KUKA KRL program: MyProgram_028().src

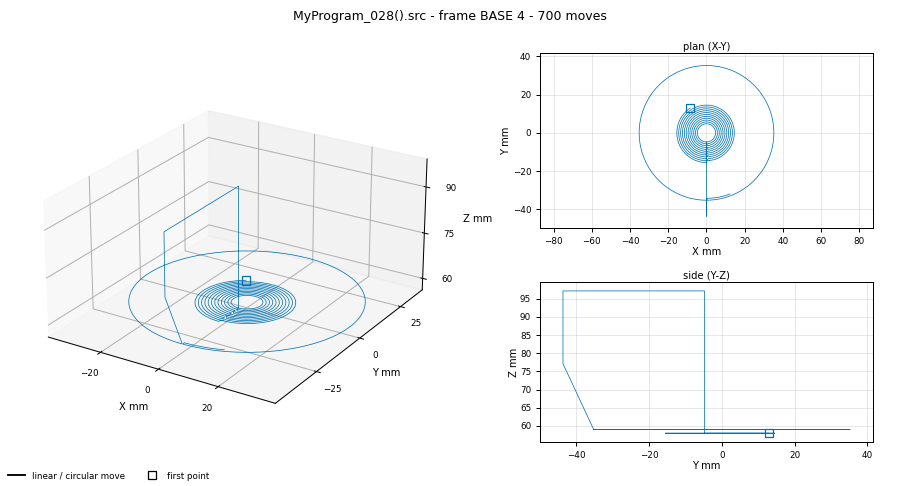
[picture p0: tool path of MyProgram_028().src in frame BASE 4, 700 of 700 moves have a stored position in this frame; points joined in program order, loops and branches not executed]
&ACCESS RVP
&REL 1
&PARAM TEMPLATE = C:\KRC\Roboter\Template\vorgabe
&PARAM EDITMASK = *
DEF MyProgram_028()
; ---- Setting reference (Base) ----
$BASE = BASE_DATA[4]

; --------------------------
; ---- Setting tool (TCP) ----
$TOOL = TOOL_DATA[3]
; --------------------------

$VEL.CP = VEL_APROX_PRINT
Startdeposition()
$VEL.CP = VEL_PRINT
LIN {X -8.4592,Y 13.0217,Z 58,A 116.025,B 24.784,C -3.3884,E1 24.9104,E2 -753.7985} C_DIS
LIN {X -9.3436,Y 12.4024,Z 58,A 119.821,B 24.785,C -3.3799,E1 24.9019,E2 -757.5875} C_DIS
LIN {X -10.555,Y 11.389,Z 58,A 127.1275,B 24.7861,C -3.3714,E1 24.8866,E2 -764.9027} C_DIS
LIN {X -12.1449,Y 9.676,Z 58,A 134.8717,B 24.7891,C -3.3477,E1 24.8724,E2 -772.6251} C_DIS
LIN {X -13.0597,Y 8.4004,Z 58,A 140.8782,B 24.791,C -3.3327,E1 24.863,E2 -778.6255} C_DIS
LIN {X -13.884,Y 6.9533,Z 58,A 146.3826,B 24.7934,C -3.3139,E1 24.8557,E2 -784.1139} C_DIS
LIN {X -14.682,Y 5.0559,Z 58,A 155.4146,B 24.7958,C -3.2945,E1 24.8466,E2 -793.15} C_DIS
LIN {X -15.1263,Y 3.5095,Z 58,A 161.5489,B 24.798,C -3.2767,E1 24.8426,E2 -799.2776} C_DIS
LIN {X -15.4979,Y 0.9698,Z 58,A 169.6776,B 24.802,C -3.2445,E1 24.8399,E2 -807.3778} C_DIS
LIN {X -15.5094,Y -0.7577,Z 58,A 177.1766,B 24.8041,C -3.2271,E1 24.8404,E2 -814.8801} C_DIS
LIN {X -15.3304,Y -2.4669,Z 58,A -177.0699,B 24.8066,C -3.2065,E1 24.8425,E2 -820.6186} C_DIS
LIN {X -14.8807,Y -4.4363,Z 58,A -169.0653,B 24.8091,C -3.1857,E1 24.8481,E2 -828.62} C_DIS
LIN {X -14.2177,Y -6.2434,Z 58,A -162.5125,B 24.8117,C -3.1645,E1 24.8549,E2 -835.1585} C_DIS
LIN {X -13.5937,Y -7.5059,Z 58,A -157.2385,B 24.8133,C -3.1509,E1 24.8617,E2 -840.428} C_DIS
LIN {X -13.0703,Y -8.3838,Z 58,A -153.3581,B 24.8144,C -3.1417,E1 24.8675,E2 -844.3061} C_DIS
LIN {X -12.191,Y -9.6177,Z 58,A -147.9234,B 24.816,C -3.1281,E1 24.8765,E2 -849.7344} C_DIS
LIN {X -11.3344,Y -10.6139,Z 58,A -142.9296,B 24.8172,C -3.1181,E1 24.8859,E2 -854.7263} C_DIS
LIN {X -10.3849,Y -11.5443,Z 58,A -138.2574,B 24.8184,C -3.1077,E1 24.8954,E2 -859.3928} C_DIS
LIN {X -9.5042,Y -12.2798,Z 58,A -134.1021,B 24.8193,C -3.0999,E1 24.9044,E2 -863.5451} C_DIS
LIN {X -8.6459,Y -12.8987,Z 58,A -129.7163,B 24.8199,C -3.0955,E1 24.9145,E2 -867.9351} C_DIS
LIN {X -7.2387,Y -13.7372,Z 58,A -123.8287,B 24.8209,C -3.0868,E1 24.9288,E2 -873.8193} C_DIS
LIN {X -5.9661,Y -14.3362,Z 58,A -119.1209,B 24.8217,C -3.0793,E1 24.9408,E2 -878.5205} C_DIS
LIN {X -4.8871,Y -14.7392,Z 58,A -114.3265,B 24.8219,C -3.0782,E1 24.9534,E2 -883.3216} C_DIS
LIN {X -3.7292,Y -15.0736,Z 58,A -110.1391,B 24.8223,C -3.0744,E1 24.9647,E2 -887.5063} C_DIS
LIN {X -2.6637,Y -15.298,Z 58,A -106.0151,B 24.8224,C -3.0735,E1 24.976,E2 -891.6326} C_DIS
LIN {X -1.431,Y -15.462,Z 58,A -101.5005,B 24.8225,C -3.0725,E1 24.9885,E2 -896.1478} C_DIS
LIN {X -0.1238,Y -15.5276,Z 58,A -96.4869,B 24.8223,C -3.0741,E1 25.0026,E2 -901.166} C_DIS
LIN {X -0.1238,Y -15.5276,Z 58,A -96.4869,B 24.8223,C -3.0741,E1 25.0026,E2 -901.166} C_DIS
Enddeposition()
LIN {X 0.0388,Y -14.5401,Z 58,A -3.2619,B 0,C 0,E1 0.1598,E2 -989.9292} C_DIS
Startdeposition()
$VEL.CP = VEL_PRINT
LIN {X -0.9942,Y -14.5149,Z 58,A -3.299,B 0,C 0,E1 0.1598,E2 -989.9288} C_DIS
LIN {X -2.6115,Y -14.3127,Z 58,A -3.3494,B 0,C 0,E1 0.1598,E2 -989.9289} C_DIS
LIN {X -4.0303,Y -13.9797,Z 58,A -3.3871,B 0,C 0,E1 0.1598,E2 -989.929} C_DIS
LIN {X -5.6828,Y -13.3931,Z 58,A -3.4223,B 0,C 0,E1 0.1598,E2 -989.9292} C_DIS
LIN {X -6.9637,Y -12.7741,Z 58,A -3.4428,B 0,C 0,E1 0.1598,E2 -989.9292} C_DIS
LIN {X -7.8731,Y -12.2346,Z 58,A -3.4532,B 0,C 0,E1 0.1598,E2 -989.9292} C_DIS
LIN {X -8.8006,Y -11.5856,Z 58,A -3.4594,B 0,C 0,E1 0.1598,E2 -989.9292} C_DIS
LIN {X -9.7294,Y -10.8172,Z 58,A -3.4607,B 0,C 0,E1 0.1598,E2 -989.9293} C_DIS
LIN {X -10.709,Y -9.8483,Z 58,A -3.4553,B 0,C 0,E1 0.1598,E2 -989.9295} C_DIS
LIN {X -11.4555,Y -8.9691,Z 58,A -3.4453,B 0,C 0,E1 0.1598,E2 -989.9295} C_DIS
LIN {X -12.3224,Y -7.735,Z 58,A -3.4244,B 0,C 0,E1 0.1598,E2 -989.9298} C_DIS
LIN {X -12.8548,Y -6.8137,Z 58,A -3.405,B 0,C 0,E1 0.1598,E2 -989.9296} C_DIS
LIN {X -13.4241,Y -5.6094,Z 58,A -3.3749,B 0,C 0,E1 0.1598,E2 -989.9296} C_DIS
LIN {X -13.7652,Y -4.7105,Z 58,A -3.3496,B 0,C 0,E1 0.1598,E2 -989.9293} C_DIS
LIN {X -14.1358,Y -3.4425,Z 58,A -3.3092,B 0,C 0,E1 0.1598,E2 -989.9297} C_DIS
LIN {X -14.3481,Y -2.4084,Z 58,A -3.2735,B 0,C 0,E1 0.1598,E2 -989.9294} C_DIS
LIN {X -14.5106,Y -1.0563,Z 58,A -3.222,B 0,C 0,E1 0.1598,E2 -989.9296} C_DIS
LIN {X -14.5449,Y 0.3484,Z 58,A -3.1636,B 0,C 0,E1 0.1598,E2 -989.9298} C_DIS
LIN {X -14.4218,Y 1.9199,Z 58,A -3.0926,B 0,C 0,E1 0.1598,E2 -989.9298} C_DIS
LIN {X -14.1478,Y 3.3932,Z 58,A -3.0205,B 0,C 0,E1 0.1598,E2 -989.9295} C_DIS
LIN {X -13.7525,Y 4.7484,Z 58,A -2.9488,B 0,C 0,E1 0.1598,E2 -989.9293} C_DIS
LIN {X -13.1379,Y 6.2501,Z 58,A -2.8624,B 0,C 0,E1 0.1598,E2 -989.9296} C_DIS
LIN {X -12.3406,Y 7.706,Z 58,A -2.7718,B 0,C 0,E1 0.1598,E2 -989.9291} C_DIS
LIN {X -11.6841,Y 8.6682,Z 58,A -2.7074,B 0,C 0,E1 0.1598,E2 -989.9285} C_DIS
LIN {X -10.8295,Y 9.7157,Z 58,A -2.6316,B 0,C 0,E1 0.1598,E2 -989.9285} C_DIS
LIN {X -10.0623,Y 10.5075,Z 58,A -2.57,B 0,C 0,E1 0.1598,E2 -989.9282} C_DIS
LIN {X -9.0076,Y 11.4252,Z 58,A -2.4922,B 0,C 0,E1 0.1598,E2 -989.9282} C_DIS
LIN {X -8.1523,Y 12.0501,Z 58,A -2.4343,B 0,C 0,E1 0.1598,E2 -989.9279} C_DIS
LIN {X -6.8933,Y 12.8124,Z 58,A -2.3555,B 0,C 0,E1 0.1598,E2 -989.9279} C_DIS
LIN {X -4.9769,Y 13.6712,Z 58,A -2.2483,B 0,C 0,E1 0.1598,E2 -989.9276} C_DIS
LIN {X -3.235,Y 14.1848,Z 58,A -2.1622,B 0,C 0,E1 0.1598,E2 -989.9274} C_DIS
LIN {X -1.6001,Y 14.4606,Z 58,A -2.09,B 0,C 0,E1 0.1598,E2 -989.9273} C_DIS
LIN {X 0.9482,Y 14.518,Z 58,A -1.9933,B 0,C 0,E1 0.1598,E2 -989.9271} C_DIS
LIN {X 1.9003,Y 14.4243,Z 58,A -1.962,B 0,C 0,E1 0.1598,E2 -989.9271} C_DIS
LIN {X 3.5313,Y 14.114,Z 58,A -1.9147,B 0,C 0,E1 0.1598,E2 -989.9271} C_DIS
LIN {X 4.9251,Y 13.6899,Z 58,A -1.8811,B 0,C 0,E1 0.1598,E2 -989.9271} C_DIS
LIN {X 6.3243,Y 13.1023,Z 58,A -1.8542,B 0,C 0,E1 0.1598,E2 -989.9272} C_DIS
LIN {X 7.3749,Y 12.5407,Z 58,A -1.8393,B 0,C 0,E1 0.1598,E2 -989.9272} C_DIS
LIN {X 8.2076,Y 12.0129,Z 58,A -1.8311,B 0,C 0,E1 0.1598,E2 -989.9271} C_DIS
LIN {X 9.0246,Y 11.4118,Z 58,A -1.8265,B 0,C 0,E1 0.1598,E2 -989.9271} C_DIS
LIN {X 10.1139,Y 10.4585,Z 58,A -1.8265,B 0,C 0,E1 0.1598,E2 -989.9275} C_DIS
LIN {X 11.0798,Y 9.4291,Z 58,A -1.8348,B 0,C 0,E1 0.1598,E2 -989.9276} C_DIS
LIN {X 11.7038,Y 8.6426,Z 58,A -1.8456,B 0,C 0,E1 0.1598,E2 -989.9273} C_DIS
LIN {X 12.3735,Y 7.6532,Z 58,A -1.8631,B 0,C 0,E1 0.1598,E2 -989.9275} C_DIS
LIN {X 13.2023,Y 6.1131,Z 58,A -1.8975,B 0,C 0,E1 0.1598,E2 -989.9285} C_DIS
LIN {X 13.7467,Y 4.7638,Z 58,A -1.9355,B 0,C 0,E1 0.1598,E2 -989.9283} C_DIS
LIN {X 14.1968,Y 3.1829,Z 58,A -1.9865,B 0,C 0,E1 0.1598,E2 -989.9286} C_DIS
LIN {X 14.3842,Y 2.1828,Z 58,A -2.0233,B 0,C 0,E1 0.1598,E2 -989.9278} C_DIS
LIN {X 14.5141,Y 1.0069,Z 58,A -2.0688,B 0,C 0,E1 0.1598,E2 -989.928} C_DIS
LIN {X 14.5491,Y -0.1159,Z 58,A -2.1158,B 0,C 0,E1 0.1598,E2 -989.928} C_DIS
LIN {X 14.4896,Y -1.3124,Z 58,A -2.1693,B 0,C 0,E1 0.1598,E2 -989.9281} C_DIS
LIN {X 14.3373,Y -2.4736,Z 58,A -2.2248,B 0,C 0,E1 0.1598,E2 -989.9281} C_DIS
LIN {X 14.0339,Y -3.8372,Z 58,A -2.2941,B 0,C 0,E1 0.1598,E2 -989.9287} C_DIS
LIN {X 13.6044,Y -5.1566,Z 58,A -2.3662,B 0,C 0,E1 0.1598,E2 -989.929} C_DIS
LIN {X 12.9068,Y -6.7148,Z 58,A -2.4589,B 0,C 0,E1 0.1598,E2 -989.929} C_DIS
LIN {X 12.2499,Y -7.8494,Z 58,A -2.5322,B 0,C 0,E1 0.1598,E2 -989.9286} C_DIS
LIN {X 11.5407,Y -8.8591,Z 58,A -2.6018,B 0,C 0,E1 0.1598,E2 -989.9284} C_DIS
LIN {X 10.8727,Y -9.6672,Z 58,A -2.6611,B 0,C 0,E1 0.1598,E2 -989.9284} C_DIS
LIN {X 9.8554,Y -10.7025,Z 58,A -2.7426,B 0,C 0,E1 0.1598,E2 -989.9286} C_DIS
LIN {X 8.7875,Y -11.5949,Z 58,A -2.8201,B 0,C 0,E1 0.1598,E2 -989.9286} C_DIS
LIN {X 7.8619,Y -12.2418,Z 58,A -2.8819,B 0,C 0,E1 0.1598,E2 -989.9285} C_DIS
LIN {X 6.6936,Y -12.918,Z 58,A -2.9536,B 0,C 0,E1 0.1598,E2 -989.9286} C_DIS
LIN {X 5.5443,Y -13.4512,Z 58,A -3.0186,B 0,C 0,E1 0.1598,E2 -989.9286} C_DIS
LIN {X 4.2078,Y -13.9272,Z 58,A -3.0879,B 0,C 0,E1 0.1598,E2 -989.9286} C_DIS
LIN {X 2.8277,Y -14.2717,Z 58,A -3.1531,B 0,C 0,E1 0.1598,E2 -989.9286} C_DIS
LIN {X 1.6425,Y -14.456,Z 58,A -3.2043,B 0,C 0,E1 0.1598,E2 -989.9287} C_DIS
LIN {X 0.0388,Y -14.5401,Z 58,A -3.2665,B 0,C 0,E1 0.1598,E2 -989.9287} C_DIS
Enddeposition()
LIN {X 0.0388,Y -14.5401,Z 58,A -3.2665,B 0,C 0,E1 0.1598,E2 -989.9287} C_DIS
Startdeposition()
$VEL.CP = VEL_PRINT
LIN {X 0.8886,Y -13.5406,Z 58,A -3.1918,B 0,C 0,E1 0.1598,E2 -989.9293} C_DIS
LIN {X 3.2193,Y -13.1824,Z 58,A -3.0918,B 0,C 0,E1 0.1598,E2 -989.9286} C_DIS
LIN {X 4.9417,Y -12.638,Z 58,A -3.0054,B 0,C 0,E1 0.1598,E2 -989.9286} C_DIS
LIN {X 6.7484,Y -11.7728,Z 58,A -2.902,B 0,C 0,E1 0.1598,E2 -989.9286} C_DIS
LIN {X 7.9074,Y -11.0278,Z 58,A -2.8277,B 0,C 0,E1 0.1598,E2 -989.9286} C_DIS
LIN {X 9.1575,Y -10.014,Z 58,A -2.7383,B 0,C 0,E1 0.1598,E2 -989.9286} C_DIS
LIN {X 10.2881,Y -8.8486,Z 58,A -2.6466,B 0,C 0,E1 0.1598,E2 -989.9287} C_DIS
LIN {X 11.189,Y -7.6776,Z 58,A -2.5634,B 0,C 0,E1 0.1598,E2 -989.9285} C_DIS
LIN {X 12.0375,Y -6.2635,Z 58,A -2.4712,B 0,C 0,E1 0.1598,E2 -989.9288} C_DIS
LIN {X 12.5414,Y -5.181,Z 58,A -2.4065,B 0,C 0,E1 0.1598,E2 -989.9284} C_DIS
LIN {X 13.1248,Y -3.4468,Z 58,A -2.3098,B 0,C 0,E1 0.1598,E2 -989.9292} C_DIS
LIN {X 13.4758,Y -1.5941,Z 58,A -2.2168,B 0,C 0,E1 0.1598,E2 -989.9296} C_DIS
LIN {X 13.4758,Y -1.5941,Z 58,A -2.2178,B 0,C 0,E1 0.1598,E2 -989.9285} C_DIS
LIN {X 13.57,Y 0.0222,Z 58,A -2.1447,B 0,C 0,E1 0.1598,E2 -989.9287} C_DIS
LIN {X 13.4778,Y 1.5775,Z 58,A -2.0812,B 0,C 0,E1 0.1598,E2 -989.9288} C_DIS
LIN {X 13.2328,Y 3.0058,Z 58,A -2.0294,B 0,C 0,E1 0.1598,E2 -989.9283} C_DIS
LIN {X 12.7101,Y 4.7521,Z 58,A -1.9731,B 0,C 0,E1 0.1598,E2 -989.9289} C_DIS
LIN {X 12.2201,Y 5.8998,Z 58,A -1.943,B 0,C 0,E1 0.1598,E2 -989.9279} C_DIS
LIN {X 11.7305,Y 6.822,Z 58,A -1.9218,B 0,C 0,E1 0.1598,E2 -989.9276} C_DIS
LIN {X 10.999,Y 7.9474,Z 58,A -1.9004,B 0,C 0,E1 0.1598,E2 -989.9278} C_DIS
LIN {X 10.0869,Y 9.0771,Z 58,A -1.8858,B 0,C 0,E1 0.1598,E2 -989.9278} C_DIS
LIN {X 9.1239,Y 10.0413,Z 58,A -1.8804,B 0,C 0,E1 0.1598,E2 -989.9276} C_DIS
LIN {X 8.0971,Y 10.8894,Z 58,A -1.8822,B 0,C 0,E1 0.1598,E2 -989.9274} C_DIS
LIN {X 7.1861,Y 11.5108,Z 58,A -1.8896,B 0,C 0,E1 0.1598,E2 -989.9272} C_DIS
LIN {X 6.149,Y 12.0958,Z 58,A -1.9031,B 0,C 0,E1 0.1598,E2 -989.9272} C_DIS
LIN {X 5.1555,Y 12.5523,Z 58,A -1.9204,B 0,C 0,E1 0.1598,E2 -989.9272} C_DIS
LIN {X 3.88,Y 13.0033,Z 58,A -1.9484,B 0,C 0,E1 0.1598,E2 -989.9272} C_DIS
LIN {X 2.4255,Y 13.3513,Z 58,A -1.9875,B 0,C 0,E1 0.1598,E2 -989.9272} C_DIS
LIN {X 1.2335,Y 13.5136,Z 58,A -2.0248,B 0,C 0,E1 0.1598,E2 -989.9272} C_DIS
LIN {X 0.0205,Y 13.5698,Z 58,A -2.0673,B 0,C 0,E1 0.1598,E2 -989.9272} C_DIS
LIN {X -1.423,Y 13.495,Z 58,A -2.1239,B 0,C 0,E1 0.1598,E2 -989.9272} C_DIS
LIN {X -2.9166,Y 13.2527,Z 58,A -2.1894,B 0,C 0,E1 0.1598,E2 -989.9274} C_DIS
LIN {X -4.4178,Y 12.8306,Z 58,A -2.2628,B 0,C 0,E1 0.1598,E2 -989.9275} C_DIS
LIN {X -5.6902,Y 12.3192,Z 58,A -2.3315,B 0,C 0,E1 0.1598,E2 -989.9277} C_DIS
LIN {X -7.1276,Y 11.5468,Z 58,A -2.4172,B 0,C 0,E1 0.1598,E2 -989.9279} C_DIS
LIN {X -8.359,Y 10.6897,Z 58,A -2.4988,B 0,C 0,E1 0.1598,E2 -989.9281} C_DIS
LIN {X -10.1247,Y 9.035,Z 58,A -2.6337,B 0,C 0,E1 0.1598,E2 -989.9286} C_DIS
LIN {X -11.3705,Y 7.4059,Z 58,A -2.7477,B 0,C 0,E1 0.1598,E2 -989.9295} C_DIS
LIN {X -11.9137,Y 6.4965,Z 58,A -2.807,B 0,C 0,E1 0.1598,E2 -989.9287} C_DIS
LIN {X -12.4568,Y 5.3822,Z 58,A -2.8739,B 0,C 0,E1 0.1598,E2 -989.929} C_DIS
LIN {X -12.8799,Y 4.271,Z 58,A -2.9366,B 0,C 0,E1 0.1598,E2 -989.929} C_DIS
LIN {X -13.4389,Y 1.8798,Z 58,A -3.0559,B 0,C 0,E1 0.1598,E2 -989.9313} C_DIS
LIN {X -13.4389,Y 1.8798,Z 58,A -3.0574,B 0,C 0,E1 0.1598,E2 -989.9299} C_DIS
LIN {X -13.5701,Y -0.0445,Z 58,A -3.1435,B 0,C 0,E1 0.1598,E2 -989.9299} C_DIS
LIN {X -13.3426,Y -2.4729,Z 58,A -3.2364,B 0,C 0,E1 0.1598,E2 -989.9314} C_DIS
LIN {X -13.3426,Y -2.4729,Z 58,A -3.2378,B 0,C 0,E1 0.1598,E2 -989.93} C_DIS
LIN {X -13.0748,Y -3.632,Z 58,A -3.2776,B 0,C 0,E1 0.1598,E2 -989.9295} C_DIS
LIN {X -12.4435,Y -5.4128,Z 58,A -3.3289,B 0,C 0,E1 0.1598,E2 -989.9305} C_DIS
LIN {X -11.9464,Y -6.436,Z 58,A -3.3549,B 0,C 0,E1 0.1598,E2 -989.9296} C_DIS
LIN {X -11.4777,Y -7.2392,Z 58,A -3.3721,B 0,C 0,E1 0.1598,E2 -989.9292} C_DIS
LIN {X -10.8186,Y -8.1914,Z 58,A -3.3882,B 0,C 0,E1 0.1598,E2 -989.9294} C_DIS
LIN {X -10.0004,Y -9.1723,Z 58,A -3.3998,B 0,C 0,E1 0.1598,E2 -989.9294} C_DIS
LIN {X -8.8658,Y -10.2733,Z 58,A -3.4052,B 0,C 0,E1 0.1598,E2 -989.9294} C_DIS
LIN {X -7.8194,Y -11.0904,Z 58,A -3.4016,B 0,C 0,E1 0.1598,E2 -989.9293} C_DIS
LIN {X -6.1046,Y -12.1193,Z 58,A -3.3824,B 0,C 0,E1 0.1598,E2 -989.9295} C_DIS
LIN {X -4.9242,Y -12.6447,Z 58,A -3.362,B 0,C 0,E1 0.1598,E2 -989.9291} C_DIS
LIN {X -3.8579,Y -13.0098,Z 58,A -3.3386,B 0,C 0,E1 0.1598,E2 -989.929} C_DIS
LIN {X -1.3592,Y -13.5016,Z 58,A -3.2683,B 0,C 0,E1 0.1598,E2 -989.9289} C_DIS
LIN {X -0.3554,Y -13.5648,Z 58,A -3.2344,B 0,C 0,E1 0.1598,E2 -989.9287} C_DIS
LIN {X -0.3554,Y -13.5648,Z 58,A -3.2344,B 0,C 0,E1 0.1598,E2 -989.9287} C_DIS
Enddeposition()
LIN {X 0.0583,Y -12.5898,Z 58,A -3.1759,B 0,C 0,E1 0.1598,E2 -989.93} C_DIS
Startdeposition()
$VEL.CP = VEL_PRINT
LIN {X -1.1152,Y -12.5412,Z 58,A -3.218,B 0,C 0,E1 0.1598,E2 -989.9288} C_DIS
LIN {X -2.5157,Y -12.3362,Z 58,A -3.2605,B 0,C 0,E1 0.1598,E2 -989.9288} C_DIS
LIN {X -3.6853,Y -12.0392,Z 58,A -3.2906,B 0,C 0,E1 0.1598,E2 -989.9288} C_DIS
LIN {X -4.9903,Y -11.5595,Z 58,A -3.3178,B 0,C 0,E1 0.1598,E2 -989.929} C_DIS
LIN {X -6.4135,Y -10.8344,Z 58,A -3.3389,B 0,C 0,E1 0.1598,E2 -989.9292} C_DIS
LIN {X -7.4925,Y -10.1188,Z 58,A -3.3479,B 0,C 0,E1 0.1598,E2 -989.9292} C_DIS
LIN {X -8.3401,Y -9.4323,Z 58,A -3.3498,B 0,C 0,E1 0.1598,E2 -989.9292} C_DIS
LIN {X -9.2947,Y -8.4931,Z 58,A -3.3447,B 0,C 0,E1 0.1598,E2 -989.9294} C_DIS
LIN {X -10.0403,Y -7.5973,Z 58,A -3.3341,B 0,C 0,E1 0.1598,E2 -989.9293} C_DIS
LIN {X -10.6375,Y -6.7357,Z 58,A -3.3194,B 0,C 0,E1 0.1598,E2 -989.9293} C_DIS
LIN {X -11.4083,Y -5.3268,Z 58,A -3.2871,B 0,C 0,E1 0.1598,E2 -989.93} C_DIS
LIN {X -11.9956,Y -3.8248,Z 58,A -3.2449,B 0,C 0,E1 0.1598,E2 -989.93} C_DIS
LIN {X -12.298,Y -2.6958,Z 58,A -3.2089,B 0,C 0,E1 0.1598,E2 -989.9294} C_DIS
LIN {X -12.4965,Y -1.5381,Z 58,A -3.167,B 0,C 0,E1 0.1598,E2 -989.9294} C_DIS
LIN {X -12.5734,Y -0.6576,Z 58,A -3.1331,B 0,C 0,E1 0.1598,E2 -989.929} C_DIS
LIN {X -12.5492,Y 1.0206,Z 58,A -3.0601,B 0,C 0,E1 0.1598,E2 -989.9299} C_DIS
LIN {X -12.3016,Y 2.682,Z 58,A -2.9801,B 0,C 0,E1 0.1598,E2 -989.9305} C_DIS
LIN {X -12.3016,Y 2.682,Z 58,A -2.9812,B 0,C 0,E1 0.1598,E2 -989.9294} C_DIS
LIN {X -11.7711,Y 4.4677,Z 58,A -2.8856,B 0,C 0,E1 0.1598,E2 -989.9298} C_DIS
LIN {X -10.8953,Y 6.3101,Z 58,A -2.7753,B 0,C 0,E1 0.1598,E2 -989.9298} C_DIS
LIN {X -9.9971,Y 7.6532,Z 58,A -2.686,B 0,C 0,E1 0.1598,E2 -989.929} C_DIS
LIN {X -9.045,Y 8.7585,Z 58,A -2.6046,B 0,C 0,E1 0.1598,E2 -989.9285} C_DIS
LIN {X -8.1234,Y 9.6193,Z 58,A -2.5343,B 0,C 0,E1 0.1598,E2 -989.9282} C_DIS
LIN {X -6.7121,Y 10.6518,Z 58,A -2.4386,B 0,C 0,E1 0.1598,E2 -989.928} C_DIS
LIN {X -5.3838,Y 11.3817,Z 58,A -2.3586,B 0,C 0,E1 0.1598,E2 -989.9279} C_DIS
LIN {X -2.878,Y 12.2573,Z 58,A -2.2289,B 0,C 0,E1 0.1598,E2 -989.9276} C_DIS
LIN {X -1.0584,Y 12.5461,Z 58,A -2.1495,B 0,C 0,E1 0.1598,E2 -989.9273} C_DIS
LIN {X 0.828,Y 12.5633,Z 58,A -2.079,B 0,C 0,E1 0.1598,E2 -989.9273} C_DIS
LIN {X 2.6155,Y 12.3161,Z 58,A -2.0234,B 0,C 0,E1 0.1598,E2 -989.9272} C_DIS
LIN {X 4.8078,Y 11.6367,Z 58,A -1.9711,B 0,C 0,E1 0.1598,E2 -989.9272} C_DIS
LIN {X 6.468,Y 10.8023,Z 58,A -1.945,B 0,C 0,E1 0.1598,E2 -989.9275} C_DIS
LIN {X 7.714,Y 9.9507,Z 58,A -1.9352,B 0,C 0,E1 0.1598,E2 -989.9275} C_DIS
LIN {X 8.7384,Y 9.0644,Z 58,A -1.9352,B 0,C 0,E1 0.1598,E2 -989.9275} C_DIS
LIN {X 9.5305,Y 8.2277,Z 58,A -1.9418,B 0,C 0,E1 0.1598,E2 -989.9275} C_DIS
LIN {X 10.3825,Y 7.1226,Z 58,A -1.9571,B 0,C 0,E1 0.1598,E2 -989.9279} C_DIS
LIN {X 11.1706,Y 5.8084,Z 58,A -1.984,B 0,C 0,E1 0.1598,E2 -989.9283} C_DIS
LIN {X 11.7313,Y 4.5716,Z 58,A -2.0165,B 0,C 0,E1 0.1598,E2 -989.928} C_DIS
LIN {X 12.1241,Y 3.3953,Z 58,A -2.0524,B 0,C 0,E1 0.1598,E2 -989.928} C_DIS
LIN {X 12.4715,Y 1.7265,Z 58,A -2.1099,B 0,C 0,E1 0.1598,E2 -989.9294} C_DIS
LIN {X 12.4715,Y 1.7265,Z 58,A -2.1109,B 0,C 0,E1 0.1598,E2 -989.9283} C_DIS
LIN {X 12.588,Y -0.2518,Z 58,A -2.1904,B 0,C 0,E1 0.1598,E2 -989.9294} C_DIS
LIN {X 12.588,Y -0.2518,Z 58,A -2.1915,B 0,C 0,E1 0.1598,E2 -989.9284} C_DIS
LIN {X 12.2824,Y -2.7694,Z 58,A -2.3081,B 0,C 0,E1 0.1598,E2 -989.9312} C_DIS
LIN {X 12.2824,Y -2.7694,Z 58,A -2.3099,B 0,C 0,E1 0.1598,E2 -989.9294} C_DIS
LIN {X 11.4381,Y -5.2626,Z 58,A -2.4463,B 0,C 0,E1 0.1598,E2 -989.9311} C_DIS
LIN {X 11.4381,Y -5.2626,Z 58,A -2.448,B 0,C 0,E1 0.1598,E2 -989.9294} C_DIS
LIN {X 10.6512,Y -6.714,Z 58,A -2.5394,B 0,C 0,E1 0.1598,E2 -989.9292} C_DIS
LIN {X 9.8702,Y -7.8162,Z 58,A -2.616,B 0,C 0,E1 0.1598,E2 -989.9285} C_DIS
LIN {X 8.4163,Y -9.3643,Z 58,A -2.7357,B 0,C 0,E1 0.1598,E2 -989.9287} C_DIS
LIN {X 7.6804,Y -9.9766,Z 58,A -2.7893,B 0,C 0,E1 0.1598,E2 -989.9283} C_DIS
LIN {X 6.4247,Y -10.8281,Z 58,A -2.8716,B 0,C 0,E1 0.1598,E2 -989.9286} C_DIS
LIN {X 5.0678,Y -11.5254,Z 58,A -2.9512,B 0,C 0,E1 0.1598,E2 -989.9286} C_DIS
LIN {X 4.0136,Y -11.9336,Z 58,A -3.0074,B 0,C 0,E1 0.1598,E2 -989.9286} C_DIS
LIN {X 2.0202,Y -12.4275,Z 58,A -3.1014,B 0,C 0,E1 0.1598,E2 -989.9286} C_DIS
LIN {X 0.6281,Y -12.5751,Z 58,A -3.1587,B 0,C 0,E1 0.1598,E2 -989.9286} C_DIS
LIN {X 0.6281,Y -12.5751,Z 58,A -3.1587,B 0,C 0,E1 0.1598,E2 -989.9286} C_DIS
Enddeposition()
LIN {X 0.0659,Y -11.608,Z 58,A -3.1363,B 0,C 0,E1 0.1598,E2 -989.9299} C_DIS
Startdeposition()
$VEL.CP = VEL_PRINT
LIN {X 0.9358,Y -11.5737,Z 58,A -3.1043,B 0,C 0,E1 0.1598,E2 -989.9286} C_DIS
LIN {X 2.2027,Y -11.4005,Z 58,A -3.0506,B 0,C 0,E1 0.1598,E2 -989.9286} C_DIS
LIN {X 3.2368,Y -11.1509,Z 58,A -3.0021,B 0,C 0,E1 0.1598,E2 -989.9285} C_DIS
LIN {X 5.2781,Y -10.3423,Z 58,A -2.8926,B 0,C 0,E1 0.1598,E2 -989.9285} C_DIS
LIN {X 6.1433,Y -9.8531,Z 58,A -2.84,B 0,C 0,E1 0.1598,E2 -989.9283} C_DIS
LIN {X 7.1677,Y -9.1352,Z 58,A -2.7715,B 0,C 0,E1 0.1598,E2 -989.9285} C_DIS
LIN {X 8.2194,Y -8.2017,Z 58,A -2.6929,B 0,C 0,E1 0.1598,E2 -989.9285} C_DIS
LIN {X 9.05,Y -7.275,Z 58,A -2.6227,B 0,C 0,E1 0.1598,E2 -989.9284} C_DIS
LIN {X 9.8561,Y -6.1384,Z 58,A -2.5441,B 0,C 0,E1 0.1598,E2 -989.9286} C_DIS
LIN {X 10.3697,Y -5.2247,Z 58,A -2.4863,B 0,C 0,E1 0.1598,E2 -989.9282} C_DIS
LIN {X 10.9795,Y -3.7785,Z 58,A -2.4013,B 0,C 0,E1 0.1598,E2 -989.9288} C_DIS
LIN {X 11.3407,Y -2.492,Z 58,A -2.3331,B 0,C 0,E1 0.1598,E2 -989.9284} C_DIS
LIN {X 11.5401,Y -1.2855,Z 58,A -2.2741,B 0,C 0,E1 0.1598,E2 -989.9283} C_DIS
LIN {X 11.6111,Y -0.1232,Z 58,A -2.2217,B 0,C 0,E1 0.1598,E2 -989.9282} C_DIS
LIN {X 11.5726,Y 0.948,Z 58,A -2.1772,B 0,C 0,E1 0.1598,E2 -989.9282} C_DIS
LIN {X 11.4265,Y 2.0639,Z 58,A -2.1348,B 0,C 0,E1 0.1598,E2 -989.928} C_DIS
LIN {X 11.1563,Y 3.2192,Z 58,A -2.0952,B 0,C 0,E1 0.1598,E2 -989.928} C_DIS
LIN {X 10.5769,Y 4.7912,Z 58,A -2.0486,B 0,C 0,E1 0.1598,E2 -989.9286} C_DIS
LIN {X 9.8604,Y 6.1315,Z 58,A -2.0179,B 0,C 0,E1 0.1598,E2 -989.9283} C_DIS
LIN {X 8.9529,Y 7.394,Z 58,A -1.9975,B 0,C 0,E1 0.1598,E2 -989.9282} C_DIS
LIN {X 8.0596,Y 8.3584,Z 58,A -1.9898,B 0,C 0,E1 0.1598,E2 -989.9277} C_DIS
LIN {X 7.0675,Y 9.2128,Z 58,A -1.9901,B 0,C 0,E1 0.1598,E2 -989.9276} C_DIS
LIN {X 5.8926,Y 10.0051,Z 58,A -1.9997,B 0,C 0,E1 0.1598,E2 -989.9275} C_DIS
LIN {X 5.0221,Y 10.4692,Z 58,A -2.0124,B 0,C 0,E1 0.1598,E2 -989.9273} C_DIS
LIN {X 4.0673,Y 10.8757,Z 58,A -2.0304,B 0,C 0,E1 0.1598,E2 -989.9273} C_DIS
LIN {X 2.8081,Y 11.2667,Z 58,A -2.0603,B 0,C 0,E1 0.1598,E2 -989.9273} C_DIS
LIN {X 1.8789,Y 11.456,Z 58,A -2.0867,B 0,C 0,E1 0.1598,E2 -989.9273} C_DIS
LIN {X 1.1267,Y 11.5541,Z 58,A -2.1104,B 0,C 0,E1 0.1598,E2 -989.9273} C_DIS
LIN {X -0.1376,Y 11.6107,Z 58,A -2.1547,B 0,C 0,E1 0.1598,E2 -989.9273} C_DIS
LIN {X -2.0552,Y 11.4281,Z 58,A -2.2333,B 0,C 0,E1 0.1598,E2 -989.9274} C_DIS
LIN {X -3.6219,Y 11.0322,Z 58,A -2.308,B 0,C 0,E1 0.1598,E2 -989.9276} C_DIS
LIN {X -5.0899,Y 10.4365,Z 58,A -2.3874,B 0,C 0,E1 0.1598,E2 -989.9278} C_DIS
LIN {X -6.3171,Y 9.7423,Z 58,A -2.462,B 0,C 0,E1 0.1598,E2 -989.928} C_DIS
LIN {X -7.671,Y 8.7161,Z 58,A -2.5551,B 0,C 0,E1 0.1598,E2 -989.9284} C_DIS
LIN {X -8.9876,Y 7.3509,Z 58,A -2.6612,B 0,C 0,E1 0.1598,E2 -989.9288} C_DIS
LIN {X -10.1678,Y 5.6075,Z 58,A -2.7778,B 0,C 0,E1 0.1598,E2 -989.9297} C_DIS
LIN {X -10.6295,Y 4.6732,Z 58,A -2.8353,B 0,C 0,E1 0.1598,E2 -989.9287} C_DIS
LIN {X -10.9996,Y 3.7108,Z 58,A -2.8897,B 0,C 0,E1 0.1598,E2 -989.9287} C_DIS
LIN {X -11.367,Y 2.3701,Z 58,A -2.9594,B 0,C 0,E1 0.1598,E2 -989.9294} C_DIS
LIN {X -11.5634,Y 1.0517,Z 58,A -3.0225,B 0,C 0,E1 0.1598,E2 -989.9294} C_DIS
LIN {X -11.5968,Y -0.5835,Z 58,A -3.0924,B 0,C 0,E1 0.1598,E2 -989.9299} C_DIS
LIN {X -11.4579,Y -1.8811,Z 58,A -3.1426,B 0,C 0,E1 0.1598,E2 -989.9295} C_DIS
LIN {X -10.93,Y -3.9197,Z 58,A -3.2094,B 0,C 0,E1 0.1598,E2 -989.9297} C_DIS
LIN {X -10.1671,Y -5.6087,Z 58,A -3.2527,B 0,C 0,E1 0.1598,E2 -989.9301} C_DIS
LIN {X -9.4269,Y -6.7795,Z 58,A -3.2758,B 0,C 0,E1 0.1598,E2 -989.9295} C_DIS
LIN {X -8.6887,Y -7.7029,Z 58,A -3.2881,B 0,C 0,E1 0.1598,E2 -989.9295} C_DIS
LIN {X -7.6348,Y -8.7484,Z 58,A -3.2939,B 0,C 0,E1 0.1598,E2 -989.9294} C_DIS
LIN {X -6.6824,Y -9.4959,Z 58,A -3.2911,B 0,C 0,E1 0.1598,E2 -989.9291} C_DIS
LIN {X -5.4334,Y -10.2618,Z 58,A -3.2779,B 0,C 0,E1 0.1598,E2 -989.9291} C_DIS
LIN {X -4.3888,Y -10.7501,Z 58,A -3.2606,B 0,C 0,E1 0.1598,E2 -989.929} C_DIS
LIN {X -3.3702,Y -11.1117,Z 58,A -3.2388,B 0,C 0,E1 0.1598,E2 -989.9288} C_DIS
LIN {X -1.4769,Y -11.5171,Z 58,A -3.1868,B 0,C 0,E1 0.1598,E2 -989.9288} C_DIS
LIN {X -0.5139,Y -11.5974,Z 58,A -3.1551,B 0,C 0,E1 0.1598,E2 -989.9286} C_DIS
LIN {X -0.5139,Y -11.5974,Z 58,A -3.1551,B 0,C 0,E1 0.1598,E2 -989.9286} C_DIS
Enddeposition()
LIN {X 0.0689,Y -10.6297,Z 58,A -3.0908,B 0,C 0,E1 0.1598,E2 -989.9299} C_DIS
Startdeposition()
$VEL.CP = VEL_PRINT
LIN {X -1.1138,Y -10.5738,Z 58,A -3.133,B 0,C 0,E1 0.1598,E2 -989.9287} C_DIS
LIN {X -2.3366,Y -10.3695,Z 58,A -3.1691,B 0,C 0,E1 0.1598,E2 -989.9287} C_DIS
LIN {X -3.1763,Y -10.1468,Z 58,A -3.1903,B 0,C 0,E1 0.1598,E2 -989.9287} C_DIS
LIN {X -4.3953,Y -9.6813,Z 58,A -3.215,B 0,C 0,E1 0.1598,E2 -989.9288} C_DIS
LIN {X -5.5525,Y -9.0673,Z 58,A -3.2312,B 0,C 0,E1 0.1598,E2 -989.9289} C_DIS
LIN {X -6.4304,Y -8.4673,Z 58,A -3.2378,B 0,C 0,E1 0.1598,E2 -989.9289} C_DIS
LIN {X -7.3345,Y -7.6976,Z 58,A -3.2381,B 0,C 0,E1 0.1598,E2 -989.9291} C_DIS
LIN {X -8.4849,Y -6.4072,Z 58,A -3.2253,B 0,C 0,E1 0.1598,E2 -989.9292} C_DIS
LIN {X -9.0728,Y -5.5434,Z 58,A -3.21,B 0,C 0,E1 0.1598,E2 -989.9294} C_DIS
LIN {X -9.7569,Y -4.2247,Z 58,A -3.1789,B 0,C 0,E1 0.1598,E2 -989.9296} C_DIS
LIN {X -10.1537,Y -3.1538,Z 58,A -3.1484,B 0,C 0,E1 0.1598,E2 -989.9292} C_DIS
LIN {X -10.4297,Y -2.0648,Z 58,A -3.1124,B 0,C 0,E1 0.1598,E2 -989.9292} C_DIS
LIN {X -10.5922,Y -0.9234,Z 58,A -3.0698,B 0,C 0,E1 0.1598,E2 -989.9293} C_DIS
LIN {X -10.6324,Y 0.0112,Z 58,A -3.0321,B 0,C 0,E1 0.1598,E2 -989.9289} C_DIS
LIN {X -10.5469,Y 1.3416,Z 58,A -2.9721,B 0,C 0,E1 0.1598,E2 -989.9293} C_DIS
LIN {X -10.3722,Y 2.3358,Z 58,A -2.924,B 0,C 0,E1 0.1598,E2 -989.9289} C_DIS
LIN {X -10.0307,Y 3.5256,Z 58,A -2.8609,B 0,C 0,E1 0.1598,E2 -989.9289} C_DIS
LIN {X -9.4167,Y 4.9368,Z 58,A -2.7781,B 0,C 0,E1 0.1598,E2 -989.9293} C_DIS
LIN {X -8.0269,Y 6.9724,Z 58,A -2.6409,B 0,C 0,E1 0.1598,E2 -989.9289} C_DIS
LIN {X -6.7605,Y 8.2055,Z 58,A -2.5421,B 0,C 0,E1 0.1598,E2 -989.9286} C_DIS
LIN {X -6.013,Y 8.7688,Z 58,A -2.4912,B 0,C 0,E1 0.1598,E2 -989.928} C_DIS
LIN {X -5.2827,Y 9.227,Z 58,A -2.4449,B 0,C 0,E1 0.1598,E2 -989.9279} C_DIS
LIN {X -3.9678,Y 9.8643,Z 58,A -2.3693,B 0,C 0,E1 0.1598,E2 -989.9279} C_DIS
LIN {X -2.6913,Y 10.286,Z 58,A -2.3043,B 0,C 0,E1 0.1598,E2 -989.9276} C_DIS
LIN {X -1.198,Y 10.5646,Z 58,A -2.2374,B 0,C 0,E1 0.1598,E2 -989.9274} C_DIS
LIN {X 0.2712,Y 10.6289,Z 58,A -2.1804,B 0,C 0,E1 0.1598,E2 -989.9274} C_DIS
LIN {X 1.5071,Y 10.5226,Z 58,A -2.1392,B 0,C 0,E1 0.1598,E2 -989.9274} C_DIS
LIN {X 2.8024,Y 10.2563,Z 58,A -2.1026,B 0,C 0,E1 0.1598,E2 -989.9274} C_DIS
LIN {X 3.8876,Y 9.896,Z 58,A -2.0778,B 0,C 0,E1 0.1598,E2 -989.9274} C_DIS
LIN {X 4.702,Y 9.5359,Z 58,A -2.0631,B 0,C 0,E1 0.1598,E2 -989.9273} C_DIS
LIN {X 5.8089,Y 8.9053,Z 58,A -2.0489,B 0,C 0,E1 0.1598,E2 -989.9274} C_DIS
LIN {X 6.8841,Y 8.1028,Z 58,A -2.0433,B 0,C 0,E1 0.1598,E2 -989.9276} C_DIS
LIN {X 7.8782,Y 7.1403,Z 58,A -2.0475,B 0,C 0,E1 0.1598,E2 -989.9277} C_DIS
LIN {X 8.7786,Y 5.9985,Z 58,A -2.0628,B 0,C 0,E1 0.1598,E2 -989.928} C_DIS
LIN {X 9.3776,Y 5.0108,Z 58,A -2.0831,B 0,C 0,E1 0.1598,E2 -989.9279} C_DIS
LIN {X 9.74,Y 4.2636,Z 58,A -2.102,B 0,C 0,E1 0.1598,E2 -989.9276} C_DIS
LIN {X 10.3374,Y 2.4868,Z 58,A -2.1545,B 0,C 0,E1 0.1598,E2 -989.9292} C_DIS
LIN {X 10.6211,Y 0.4869,Z 58,A -2.2293,B 0,C 0,E1 0.1598,E2 -989.9297} C_DIS
LIN {X 10.6211,Y 0.4869,Z 58,A -2.2304,B 0,C 0,E1 0.1598,E2 -989.9285} C_DIS
LIN {X 10.5933,Y -0.9108,Z 58,A -2.2913,B 0,C 0,E1 0.1598,E2 -989.9286} C_DIS
LIN {X 10.4469,Y -1.9768,Z 58,A -2.3428,B 0,C 0,E1 0.1598,E2 -989.9282} C_DIS
LIN {X 10.1303,Y -3.2277,Z 58,A -2.4077,B 0,C 0,E1 0.1598,E2 -989.9287} C_DIS
LIN {X 9.6928,Y -4.3697,Z 58,A -2.473,B 0,C 0,E1 0.1598,E2 -989.9285} C_DIS
LIN {X 9.0572,Y -5.569,Z 58,A -2.5476,B 0,C 0,E1 0.1598,E2 -989.9287} C_DIS
LIN {X 8.5038,Y -6.3819,Z 58,A -2.6032,B 0,C 0,E1 0.1598,E2 -989.9282} C_DIS
LIN {X 7.0479,Y -7.9609,Z 58,A -2.7234,B 0,C 0,E1 0.1598,E2 -989.9292} C_DIS
LIN {X 5.4991,Y -9.0993,Z 58,A -2.8297,B 0,C 0,E1 0.1598,E2 -989.9285} C_DIS
LIN {X 3.9607,Y -9.867,Z 58,A -2.9191,B 0,C 0,E1 0.1598,E2 -989.9285} C_DIS
LIN {X 2.3268,Y -10.3747,Z 58,A -3.0006,B 0,C 0,E1 0.1598,E2 -989.9285} C_DIS
LIN {X 0.9025,Y -10.594,Z 58,A -3.0622,B 0,C 0,E1 0.1598,E2 -989.9285} C_DIS
LIN {X 0.0689,Y -10.6297,Z 58,A -3.0943,B 0,C 0,E1 0.1598,E2 -989.9285} C_DIS
Enddeposition()
LIN {X 0.0689,Y -10.6297,Z 58,A -3.0943,B 0,C 0,E1 0.1598,E2 -989.9285} C_DIS
Startdeposition()
$VEL.CP = VEL_PRINT
LIN {X 0.4362,Y -9.6432,Z 58,A -3.0378,B 0,C 0,E1 0.1598,E2 -989.9291} C_DIS
LIN {X 1.6154,Y -9.517,Z 58,A -2.9898,B 0,C 0,E1 0.1598,E2 -989.9285} C_DIS
LIN {X 2.5756,Y -9.3029,Z 58,A -2.9455,B 0,C 0,E1 0.1598,E2 -989.9284} C_DIS
LIN {X 4.2409,Y -8.6715,Z 58,A -2.8573,B 0,C 0,E1 0.1598,E2 -989.9284} C_DIS
LIN {X 5.3054,Y -8.0644,Z 58,A -2.7924,B 0,C 0,E1 0.1598,E2 -989.9284} C_DIS
LIN {X 6.2458,Y -7.3552,Z 58,A -2.7275,B 0,C 0,E1 0.1598,E2 -989.9284} C_DIS
LIN {X 6.8828,Y -6.7623,Z 58,A -2.6788,B 0,C 0,E1 0.1598,E2 -989.9282} C_DIS
LIN {X 7.658,Y -5.8767,Z 58,A -2.6123,B 0,C 0,E1 0.1598,E2 -989.9282} C_DIS
LIN {X 8.2664,Y -4.9848,Z 58,A -2.5517,B 0,C 0,E1 0.1598,E2 -989.9282} C_DIS
LIN {X 8.7593,Y -4.0565,Z 58,A -2.4937,B 0,C 0,E1 0.1598,E2 -989.9282} C_DIS
LIN {X 9.1308,Y -3.1327,Z 58,A -2.4406,B 0,C 0,E1 0.1598,E2 -989.9282} C_DIS
LIN {X 9.558,Y -1.3515,Z 58,A -2.3474,B 0,C 0,E1 0.1598,E2 -989.9292} C_DIS
LIN {X 9.6417,Y -0.4638,Z 58,A -2.3074,B 0,C 0,E1 0.1598,E2 -989.928} C_DIS
LIN {X 9.6313,Y 0.6472,Z 58,A -2.26,B 0,C 0,E1 0.1598,E2 -989.9282} C_DIS
LIN {X 9.5188,Y 1.6038,Z 58,A -2.2234,B 0,C 0,E1 0.1598,E2 -989.9279} C_DIS
LIN {X 9.2565,Y 2.7384,Z 58,A -2.1843,B 0,C 0,E1 0.1598,E2 -989.9281} C_DIS
LIN {X 8.7719,Y 4.0293,Z 58,A -2.1467,B 0,C 0,E1 0.1598,E2 -989.9282} C_DIS
LIN {X 8.164,Y 5.1505,Z 58,A -2.1213,B 0,C 0,E1 0.1598,E2 -989.9282} C_DIS
LIN {X 7.4711,Y 6.1094,Z 58,A -2.1061,B 0,C 0,E1 0.1598,E2 -989.9278} C_DIS
LIN {X 6.6884,Y 6.9604,Z 58,A -2.0988,B 0,C 0,E1 0.1598,E2 -989.9277} C_DIS
LIN {X 5.9421,Y 7.6076,Z 58,A -2.0989,B 0,C 0,E1 0.1598,E2 -989.9275} C_DIS
LIN {X 4.8585,Y 8.3411,Z 58,A -2.1075,B 0,C 0,E1 0.1598,E2 -989.9276} C_DIS
LIN {X 3.7731,Y 8.8851,Z 58,A -2.1246,B 0,C 0,E1 0.1598,E2 -989.9275} C_DIS
LIN {X 2.5898,Y 9.295,Z 58,A -2.1509,B 0,C 0,E1 0.1598,E2 -989.9275} C_DIS
LIN {X 1.5435,Y 9.529,Z 58,A -2.1797,B 0,C 0,E1 0.1598,E2 -989.9274} C_DIS
LIN {X 0.584,Y 9.6355,Z 58,A -2.2106,B 0,C 0,E1 0.1598,E2 -989.9274} C_DIS
LIN {X -0.667,Y 9.6299,Z 58,A -2.2571,B 0,C 0,E1 0.1598,E2 -989.9274} C_DIS
LIN {X -1.7147,Y 9.4996,Z 58,A -2.3013,B 0,C 0,E1 0.1598,E2 -989.9275} C_DIS
LIN {X -2.6436,Y 9.284,Z 58,A -2.3448,B 0,C 0,E1 0.1598,E2 -989.9275} C_DIS
LIN {X -3.778,Y 8.8831,Z 58,A -2.4036,B 0,C 0,E1 0.1598,E2 -989.9277} C_DIS
LIN {X -5.0223,Y 8.2436,Z 58,A -2.4765,B 0,C 0,E1 0.1598,E2 -989.9279} C_DIS
LIN {X -6.0733,Y 7.5028,Z 58,A -2.5466,B 0,C 0,E1 0.1598,E2 -989.9281} C_DIS
LIN {X -7.3351,Y 6.2753,Z 58,A -2.6447,B 0,C 0,E1 0.1598,E2 -989.9287} C_DIS
LIN {X -8.2,Y 5.0932,Z 58,A -2.7266,B 0,C 0,E1 0.1598,E2 -989.9288} C_DIS
LIN {X -8.7074,Y 4.167,Z 58,A -2.7848,B 0,C 0,E1 0.1598,E2 -989.9286} C_DIS
LIN {X -9.1582,Y 3.0515,Z 58,A -2.8485,B 0,C 0,E1 0.1598,E2 -989.9288} C_DIS
LIN {X -9.4962,Y 1.7335,Z 58,A -2.9164,B 0,C 0,E1 0.1598,E2 -989.9292} C_DIS
LIN {X -9.6522,Y 0.1078,Z 58,A -2.9907,B 0,C 0,E1 0.1598,E2 -989.9297} C_DIS
LIN {X -9.5814,Y -1.1756,Z 58,A -3.0422,B 0,C 0,E1 0.1598,E2 -989.93} C_DIS
LIN {X -9.2308,Y -2.8235,Z 58,A -3.0993,B 0,C 0,E1 0.1598,E2 -989.9299} C_DIS
LIN {X -8.665,Y -4.2545,Z 58,A -3.1395,B 0,C 0,E1 0.1598,E2 -989.9296} C_DIS
LIN {X -7.8201,Y -5.6597,Z 58,A -3.1682,B 0,C 0,E1 0.1598,E2 -989.9296} C_DIS
LIN {X -7.142,Y -6.4943,Z 58,A -3.1793,B 0,C 0,E1 0.1598,E2 -989.9291} C_DIS
LIN {X -5.8919,Y -7.6464,Z 58,A -3.1821,B 0,C 0,E1 0.1598,E2 -989.9294} C_DIS
LIN {X -4.7598,Y -8.398,Z 58,A -3.1731,B 0,C 0,E1 0.1598,E2 -989.929} C_DIS
LIN {X -3.6431,Y -8.9392,Z 58,A -3.1553,B 0,C 0,E1 0.1598,E2 -989.9288} C_DIS
LIN {X -1.8172,Y -9.4805,Z 58,A -3.1115,B 0,C 0,E1 0.1598,E2 -989.9288} C_DIS
LIN {X -0.2654,Y -9.6483,Z 58,A -3.062,B 0,C 0,E1 0.1598,E2 -989.9285} C_DIS
LIN {X -0.2654,Y -9.6483,Z 58,A -3.062,B 0,C 0,E1 0.1598,E2 -989.9285} C_DIS
Enddeposition()
LIN {X 0.0369,Y -8.6725,Z 58,A -3.0077,B 0,C 0,E1 0.1598,E2 -989.9298} C_DIS
Startdeposition()
$VEL.CP = VEL_PRINT
LIN {X -0.8559,Y -8.6313,Z 58,A -3.0399,B 0,C 0,E1 0.1598,E2 -989.9286} C_DIS
LIN {X -2.0086,Y -8.4381,Z 58,A -3.074,B 0,C 0,E1 0.1598,E2 -989.9286} C_DIS
LIN {X -2.8766,Y -8.183,Z 58,A -3.0949,B 0,C 0,E1 0.1598,E2 -989.9286} C_DIS
LIN {X -4.2356,Y -7.5694,Z 58,A -3.1184,B 0,C 0,E1 0.1598,E2 -989.9288} C_DIS
LIN {X -5.0287,Y -7.0626,Z 58,A -3.126,B 0,C 0,E1 0.1598,E2 -989.9288} C_DIS
LIN {X -5.6229,Y -6.6001,Z 58,A -3.1281,B 0,C 0,E1 0.1598,E2 -989.9288} C_DIS
LIN {X -6.4,Y -5.8546,Z 58,A -3.1247,B 0,C 0,E1 0.1598,E2 -989.9288} C_DIS
LIN {X -7.0818,Y -5.0086,Z 58,A -3.1137,B 0,C 0,E1 0.1598,E2 -989.929} C_DIS
LIN {X -7.7745,Y -3.8462,Z 58,A -3.0893,B 0,C 0,E1 0.1598,E2 -989.9294} C_DIS
LIN {X -8.2704,Y -2.6147,Z 58,A -3.0553,B 0,C 0,E1 0.1598,E2 -989.9294} C_DIS
LIN {X -8.5439,Y -1.4938,Z 58,A -3.0179,B 0,C 0,E1 0.1598,E2 -989.9291} C_DIS
LIN {X -8.6735,Y -0.1001,Z 58,A -2.9633,B 0,C 0,E1 0.1598,E2 -989.9294} C_DIS
LIN {X -8.601,Y 1.1227,Z 58,A -2.9088,B 0,C 0,E1 0.1598,E2 -989.9293} C_DIS
LIN {X -8.2607,Y 2.6455,Z 58,A -2.8312,B 0,C 0,E1 0.1598,E2 -989.9297} C_DIS
LIN {X -7.6866,Y 4.0187,Z 58,A -2.7525,B 0,C 0,E1 0.1598,E2 -989.929} C_DIS
LIN {X -7.2157,Y 4.8134,Z 58,A -2.7019,B 0,C 0,E1 0.1598,E2 -989.9285} C_DIS
LIN {X -6.3584,Y 5.8987,Z 58,A -2.6241,B 0,C 0,E1 0.1598,E2 -989.9285} C_DIS
LIN {X -4.8078,Y 7.2196,Z 58,A -2.5111,B 0,C 0,E1 0.1598,E2 -989.9282} C_DIS
LIN {X -3.7098,Y 7.8405,Z 58,A -2.4445,B 0,C 0,E1 0.1598,E2 -989.9279} C_DIS
LIN {X -2.5241,Y 8.2986,Z 58,A -2.3814,B 0,C 0,E1 0.1598,E2 -989.9277} C_DIS
LIN {X -1.3048,Y 8.5748,Z 58,A -2.3247,B 0,C 0,E1 0.1598,E2 -989.9276} C_DIS
LIN {X 0.0955,Y 8.6734,Z 58,A -2.2688,B 0,C 0,E1 0.1598,E2 -989.9275} C_DIS
LIN {X 1.4569,Y 8.5478,Z 58,A -2.2239,B 0,C 0,E1 0.1598,E2 -989.9275} C_DIS
LIN {X 2.5435,Y 8.2926,Z 58,A -2.1946,B 0,C 0,E1 0.1598,E2 -989.9275} C_DIS
LIN {X 3.9118,Y 7.7413,Z 58,A -2.1674,B 0,C 0,E1 0.1598,E2 -989.9275} C_DIS
LIN {X 4.8652,Y 7.181,Z 58,A -2.1561,B 0,C 0,E1 0.1598,E2 -989.9275} C_DIS
LIN {X 5.6273,Y 6.6007,Z 58,A -2.1527,B 0,C 0,E1 0.1598,E2 -989.9275} C_DIS
LIN {X 6.5461,Y 5.6849,Z 58,A -2.1576,B 0,C 0,E1 0.1598,E2 -989.9278} C_DIS
LIN {X 7.0912,Y 4.9893,Z 58,A -2.1674,B 0,C 0,E1 0.1598,E2 -989.9276} C_DIS
LIN {X 7.6708,Y 4.0491,Z 58,A -2.1859,B 0,C 0,E1 0.1598,E2 -989.928} C_DIS
LIN {X 8.1928,Y 2.8488,Z 58,A -2.2177,B 0,C 0,E1 0.1598,E2 -989.9283} C_DIS
LIN {X 8.6361,Y 0.8095,Z 58,A -2.2872,B 0,C 0,E1 0.1598,E2 -989.9298} C_DIS
LIN {X 8.6361,Y 0.8095,Z 58,A -2.2883,B 0,C 0,E1 0.1598,E2 -989.9287} C_DIS
LIN {X 8.6506,Y -0.6353,Z 58,A -2.3495,B 0,C 0,E1 0.1598,E2 -989.9287} C_DIS
LIN {X 8.4953,Y -1.7514,Z 58,A -2.4035,B 0,C 0,E1 0.1598,E2 -989.9284} C_DIS
LIN {X 8.2048,Y -2.8055,Z 58,A -2.4594,B 0,C 0,E1 0.1598,E2 -989.9284} C_DIS
LIN {X 7.9465,Y -3.4712,Z 58,A -2.4977,B 0,C 0,E1 0.1598,E2 -989.928} C_DIS
LIN {X 7.5498,Y -4.2707,Z 58,A -2.5464,B 0,C 0,E1 0.1598,E2 -989.9282} C_DIS
LIN {X 6.9763,Y -5.1543,Z 58,A -2.6052,B 0,C 0,E1 0.1598,E2 -989.9283} C_DIS
LIN {X 6.3626,Y -5.8953,Z 58,A -2.6596,B 0,C 0,E1 0.1598,E2 -989.9283} C_DIS
LIN {X 5.8293,Y -6.4232,Z 58,A -2.7019,B 0,C 0,E1 0.1598,E2 -989.9282} C_DIS
LIN {X 4.9655,Y -7.1089,Z 58,A -2.7628,B 0,C 0,E1 0.1598,E2 -989.9283} C_DIS
LIN {X 4.0218,Y -7.6852,Z 58,A -2.8221,B 0,C 0,E1 0.1598,E2 -989.9283} C_DIS
LIN {X 2.768,Y -8.2204,Z 58,A -2.8909,B 0,C 0,E1 0.1598,E2 -989.9284} C_DIS
LIN {X 1.759,Y -8.4933,Z 58,A -2.9397,B 0,C 0,E1 0.1598,E2 -989.9284} C_DIS
LIN {X 0.7467,Y -8.6415,Z 58,A -2.9831,B 0,C 0,E1 0.1598,E2 -989.9284} C_DIS
LIN {X 0.7467,Y -8.6415,Z 58,A -2.9831,B 0,C 0,E1 0.1598,E2 -989.9284} C_DIS
Enddeposition()
LIN {X 0.0421,Y -7.694,Z 58,A -2.9669,B 0,C 0,E1 0.1598,E2 -989.9297} C_DIS
Startdeposition()
$VEL.CP = VEL_PRINT
LIN {X 1.442,Y -7.5584,Z 58,A -2.9111,B 0,C 0,E1 0.1598,E2 -989.9284} C_DIS
LIN {X 2.7625,Y -7.1817,Z 58,A -2.8466,B 0,C 0,E1 0.1598,E2 -989.9283} C_DIS
LIN {X 3.4645,Y -6.8708,Z 58,A -2.8076,B 0,C 0,E1 0.1598,E2 -989.9283} C_DIS
LIN {X 4.1845,Y -6.4574,Z 58,A -2.7635,B 0,C 0,E1 0.1598,E2 -989.9282} C_DIS
LIN {X 5.1265,Y -5.7335,Z 58,A -2.6978,B 0,C 0,E1 0.1598,E2 -989.9283} C_DIS
LIN {X 5.7505,Y -5.1129,Z 58,A -2.6483,B 0,C 0,E1 0.1598,E2 -989.9283} C_DIS
LIN {X 6.4394,Y -4.2123,Z 58,A -2.5844,B 0,C 0,E1 0.1598,E2 -989.9283} C_DIS
LIN {X 7.008,Y -3.1765,Z 58,A -2.5189,B 0,C 0,E1 0.1598,E2 -989.9285} C_DIS
LIN {X 7.4045,Y -2.0931,Z 58,A -2.458,B 0,C 0,E1 0.1598,E2 -989.9283} C_DIS
LIN {X 7.6236,Y -1.0168,Z 58,A -2.404,B 0,C 0,E1 0.1598,E2 -989.9283} C_DIS
LIN {X 7.6919,Y -0.1986,Z 58,A -2.3666,B 0,C 0,E1 0.1598,E2 -989.9281} C_DIS
LIN {X 7.6309,Y 0.9891,Z 58,A -2.3177,B 0,C 0,E1 0.1598,E2 -989.9283} C_DIS
LIN {X 7.4333,Y 1.988,Z 58,A -2.2825,B 0,C 0,E1 0.1598,E2 -989.9281} C_DIS
LIN {X 7.0262,Y 3.1368,Z 58,A -2.2482,B 0,C 0,E1 0.1598,E2 -989.9282} C_DIS
LIN {X 6.5451,Y 4.0463,Z 58,A -2.2273,B 0,C 0,E1 0.1598,E2 -989.9279} C_DIS
LIN {X 5.9028,Y 4.9363,Z 58,A -2.213,B 0,C 0,E1 0.1598,E2 -989.9279} C_DIS
LIN {X 5.2297,Y 5.6444,Z 58,A -2.2078,B 0,C 0,E1 0.1598,E2 -989.9277} C_DIS
LIN {X 4.3953,Y 6.3159,Z 58,A -2.2099,B 0,C 0,E1 0.1598,E2 -989.9277} C_DIS
LIN {X 3.2343,Y 6.9816,Z 58,A -2.2244,B 0,C 0,E1 0.1598,E2 -989.9277} C_DIS
LIN {X 2.1893,Y 7.3767,Z 58,A -2.2463,B 0,C 0,E1 0.1598,E2 -989.9276} C_DIS
LIN {X 0.8793,Y 7.6441,Z 58,A -2.2833,B 0,C 0,E1 0.1598,E2 -989.9276} C_DIS
LIN {X -0.6233,Y 7.6695,Z 58,A -2.3378,B 0,C 0,E1 0.1598,E2 -989.9276} C_DIS
LIN {X -1.6138,Y 7.5237,Z 58,A -2.3805,B 0,C 0,E1 0.1598,E2 -989.9276} C_DIS
LIN {X -2.7826,Y 7.1741,Z 58,A -2.4385,B 0,C 0,E1 0.1598,E2 -989.9277} C_DIS
LIN {X -3.9293,Y 6.6151,Z 58,A -2.5044,B 0,C 0,E1 0.1598,E2 -989.9279} C_DIS
LIN {X -4.9668,Y 5.8767,Z 58,A -2.5738,B 0,C 0,E1 0.1598,E2 -989.9282} C_DIS
LIN {X -5.9937,Y 4.8206,Z 58,A -2.6562,B 0,C 0,E1 0.1598,E2 -989.9285} C_DIS
LIN {X -6.5215,Y 4.084,Z 58,A -2.7069,B 0,C 0,E1 0.1598,E2 -989.9285} C_DIS
LIN {X -7.1104,Y 2.9417,Z 58,A -2.7769,B 0,C 0,E1 0.1598,E2 -989.9288} C_DIS
LIN {X -7.5284,Y 1.5912,Z 58,A -2.8491,B 0,C 0,E1 0.1598,E2 -989.9293} C_DIS
LIN {X -7.6738,Y 0.5688,Z 58,A -2.8983,B 0,C 0,E1 0.1598,E2 -989.9289} C_DIS
LIN {X -7.6745,Y -0.549,Z 58,A -2.9456,B 0,C 0,E1 0.1598,E2 -989.9289} C_DIS
LIN {X -7.3943,Y -2.1293,Z 58,A -3.0017,B 0,C 0,E1 0.1598,E2 -989.9297} C_DIS
LIN {X -6.9282,Y -3.3477,Z 58,A -3.0365,B 0,C 0,E1 0.1598,E2 -989.9295} C_DIS
LIN {X -6.0439,Y -4.7558,Z 58,A -3.0639,B 0,C 0,E1 0.1598,E2 -989.9295} C_DIS
LIN {X -5.1969,Y -5.6746,Z 58,A -3.0724,B 0,C 0,E1 0.1598,E2 -989.929} C_DIS
LIN {X -4.4773,Y -6.2521,Z 58,A -3.0709,B 0,C 0,E1 0.1598,E2 -989.9287} C_DIS
LIN {X -3.6986,Y -6.7474,Z 58,A -3.0634,B 0,C 0,E1 0.1598,E2 -989.9287} C_DIS
LIN {X -2.1313,Y -7.3937,Z 58,A -3.0334,B 0,C 0,E1 0.1598,E2 -989.9287} C_DIS
LIN {X -0.1687,Y -7.6929,Z 58,A -2.9744,B 0,C 0,E1 0.1598,E2 -989.9285} C_DIS
LIN {X -0.1687,Y -7.6929,Z 58,A -2.9744,B 0,C 0,E1 0.1598,E2 -989.9285} C_DIS
Enddeposition()
LIN {X 0.0469,Y -6.7119,Z 58,A -2.9232,B 0,C 0,E1 0.1598,E2 -989.9297} C_DIS
Startdeposition()
$VEL.CP = VEL_PRINT
LIN {X -0.7774,Y -6.6702,Z 58,A -2.9529,B 0,C 0,E1 0.1598,E2 -989.9284} C_DIS
LIN {X -1.6075,Y -6.5174,Z 58,A -2.9768,B 0,C 0,E1 0.1598,E2 -989.9284} C_DIS
LIN {X -2.5898,Y -6.1961,Z 58,A -2.9991,B 0,C 0,E1 0.1598,E2 -989.9284} C_DIS
LIN {X -3.2648,Y -5.8654,Z 58,A -3.0098,B 0,C 0,E1 0.1598,E2 -989.9284} C_DIS
LIN {X -4.0647,Y -5.3459,Z 58,A -3.0169,B 0,C 0,E1 0.1598,E2 -989.9286} C_DIS
LIN {X -4.7991,Y -4.6977,Z 58,A -3.0163,B 0,C 0,E1 0.1598,E2 -989.9286} C_DIS
LIN {X -5.4754,Y -3.8797,Z 58,A -3.0062,B 0,C 0,E1 0.1598,E2 -989.9288} C_DIS
LIN {X -6.1314,Y -2.7395,Z 58,A -2.9813,B 0,C 0,E1 0.1598,E2 -989.9292} C_DIS
LIN {X -6.4875,Y -1.7353,Z 58,A -2.9521,B 0,C 0,E1 0.1598,E2 -989.9289} C_DIS
LIN {X -6.7117,Y -0.2283,Z 58,A -2.8956,B 0,C 0,E1 0.1598,E2 -989.9296} C_DIS
LIN {X -6.6783,Y 0.6495,Z 58,A -2.858,B 0,C 0,E1 0.1598,E2 -989.9287} C_DIS
LIN {X -6.542,Y 1.5172,Z 58,A -2.8161,B 0,C 0,E1 0.1598,E2 -989.9287} C_DIS
LIN {X -6.2744,Y 2.3937,Z 58,A -2.7692,B 0,C 0,E1 0.1598,E2 -989.9285} C_DIS
LIN {X -5.8104,Y 3.3674,Z 58,A -2.7106,B 0,C 0,E1 0.1598,E2 -989.9285} C_DIS
LIN {X -5.3339,Y 4.0801,Z 58,A -2.663,B 0,C 0,E1 0.1598,E2 -989.9283} C_DIS
LIN {X -4.8721,Y 4.6156,Z 58,A -2.6234,B 0,C 0,E1 0.1598,E2 -989.9281} C_DIS
LIN {X -4.336,Y 5.1278,Z 58,A -2.582,B 0,C 0,E1 0.1598,E2 -989.9281} C_DIS
LIN {X -3.488,Y 5.7387,Z 58,A -2.5247,B 0,C 0,E1 0.1598,E2 -989.928} C_DIS
LIN {X -2.5491,Y 6.2077,Z 58,A -2.4703,B 0,C 0,E1 0.1598,E2 -989.9278} C_DIS
LIN {X -1.5518,Y 6.5339,Z 58,A -2.4197,B 0,C 0,E1 0.1598,E2 -989.9278} C_DIS
LIN {X -0.5614,Y 6.6921,Z 58,A -2.3765,B 0,C 0,E1 0.1598,E2 -989.9276} C_DIS
LIN {X 0.9092,Y 6.6538,Z 58,A -2.3239,B 0,C 0,E1 0.1598,E2 -989.9276} C_DIS
LIN {X 2.2503,Y 6.3213,Z 58,A -2.2885,B 0,C 0,E1 0.1598,E2 -989.9276} C_DIS
LIN {X 3.2509,Y 5.8764,Z 58,A -2.2705,B 0,C 0,E1 0.1598,E2 -989.9276} C_DIS
LIN {X 4.1065,Y 5.3137,Z 58,A -2.2628,B 0,C 0,E1 0.1598,E2 -989.9276} C_DIS
LIN {X 4.8484,Y 4.6467,Z 58,A -2.2638,B 0,C 0,E1 0.1598,E2 -989.9277} C_DIS
LIN {X 5.4298,Y 3.9449,Z 58,A -2.2724,B 0,C 0,E1 0.1598,E2 -989.9277} C_DIS
LIN {X 5.8241,Y 3.3319,Z 58,A -2.284,B 0,C 0,E1 0.1598,E2 -989.9277} C_DIS
LIN {X 6.3714,Y 2.1225,Z 58,A -2.3148,B 0,C 0,E1 0.1598,E2 -989.9285} C_DIS
LIN {X 6.6667,Y 0.8042,Z 58,A -2.3603,B 0,C 0,E1 0.1598,E2 -989.9285} C_DIS
LIN {X 6.6561,Y -0.8923,Z 58,A -2.4324,B 0,C 0,E1 0.1598,E2 -989.9294} C_DIS
LIN {X 6.4289,Y -1.9402,Z 58,A -2.4864,B 0,C 0,E1 0.1598,E2 -989.9286} C_DIS
LIN {X 6.0032,Y -2.998,Z 58,A -2.5475,B 0,C 0,E1 0.1598,E2 -989.9284} C_DIS
LIN {X 5.6283,Y -3.6516,Z 58,A -2.5896,B 0,C 0,E1 0.1598,E2 -989.9281} C_DIS
LIN {X 5.1852,Y -4.261,Z 58,A -2.6319,B 0,C 0,E1 0.1598,E2 -989.9281} C_DIS
LIN {X 4.6746,Y -4.8154,Z 58,A -2.6744,B 0,C 0,E1 0.1598,E2 -989.9281} C_DIS
LIN {X 3.847,Y -5.5045,Z 58,A -2.7342,B 0,C 0,E1 0.1598,E2 -989.9283} C_DIS
LIN {X 2.5719,Y -6.2035,Z 58,A -2.8108,B 0,C 0,E1 0.1598,E2 -989.9283} C_DIS
LIN {X 1.3969,Y -6.5649,Z 58,A -2.8695,B 0,C 0,E1 0.1598,E2 -989.9283} C_DIS
LIN {X 0.6614,Y -6.683,Z 58,A -2.9015,B 0,C 0,E1 0.1598,E2 -989.9283} C_DIS
LIN {X 0.6614,Y -6.683,Z 58,A -2.9015,B 0,C 0,E1 0.1598,E2 -989.9283} C_DIS
Enddeposition()
LIN {X 0.0501,Y -5.7324,Z 58,A -2.8819,B 0,C 0,E1 0.1598,E2 -989.9296} C_DIS
Startdeposition()
$VEL.CP = VEL_PRINT
LIN {X 0.7687,Y -5.6839,Z 58,A -2.8547,B 0,C 0,E1 0.1598,E2 -989.9283} C_DIS
LIN {X 1.6613,Y -5.4906,Z 58,A -2.8138,B 0,C 0,E1 0.1598,E2 -989.9282} C_DIS
LIN {X 2.5108,Y -5.1553,Z 58,A -2.7683,B 0,C 0,E1 0.1598,E2 -989.9282} C_DIS
LIN {X 3.2101,Y -4.7506,Z 58,A -2.7253,B 0,C 0,E1 0.1598,E2 -989.9282} C_DIS
LIN {X 3.7023,Y -4.3817,Z 58,A -2.6915,B 0,C 0,E1 0.1598,E2 -989.9281} C_DIS
LIN {X 4.51,Y -3.5358,Z 58,A -2.6254,B 0,C 0,E1 0.1598,E2 -989.9283} C_DIS
LIN {X 4.9361,Y -2.91,Z 58,A -2.5831,B 0,C 0,E1 0.1598,E2 -989.9281} C_DIS
LIN {X 5.2777,Y -2.2345,Z 58,A -2.5417,B 0,C 0,E1 0.1598,E2 -989.9281} C_DIS
LIN {X 5.5272,Y -1.5196,Z 58,A -2.5019,B 0,C 0,E1 0.1598,E2 -989.9281} C_DIS
LIN {X 5.706,Y -0.5901,Z 58,A -2.4554,B 0,C 0,E1 0.1598,E2 -989.9283} C_DIS
LIN {X 5.7267,Y 0.2302,Z 58,A -2.4197,B 0,C 0,E1 0.1598,E2 -989.928} C_DIS
LIN {X 5.6622,Y 0.9171,Z 58,A -2.3929,B 0,C 0,E1 0.1598,E2 -989.9279} C_DIS
LIN {X 5.373,Y 1.997,Z 58,A -2.357,B 0,C 0,E1 0.1598,E2 -989.9282} C_DIS
LIN {X 5.0697,Y 2.674,Z 58,A -2.3396,B 0,C 0,E1 0.1598,E2 -989.9278} C_DIS
LIN {X 4.6797,Y 3.3047,Z 58,A -2.3271,B 0,C 0,E1 0.1598,E2 -989.9278} C_DIS
LIN {X 4.2153,Y 3.883,Z 58,A -2.3196,B 0,C 0,E1 0.1598,E2 -989.9278} C_DIS
LIN {X 3.6795,Y 4.3961,Z 58,A -2.3175,B 0,C 0,E1 0.1598,E2 -989.9277} C_DIS
LIN {X 3.0806,Y 4.8338,Z 58,A -2.321,B 0,C 0,E1 0.1598,E2 -989.9277} C_DIS
LIN {X 2.4297,Y 5.1893,Z 58,A -2.3299,B 0,C 0,E1 0.1598,E2 -989.9277} C_DIS
LIN {X 1.739,Y 5.4592,Z 58,A -2.3439,B 0,C 0,E1 0.1598,E2 -989.9277} C_DIS
LIN {X 0.4411,Y 5.7192,Z 58,A -2.3807,B 0,C 0,E1 0.1598,E2 -989.9277} C_DIS
LIN {X -0.6671,Y 5.6935,Z 58,A -2.4227,B 0,C 0,E1 0.1598,E2 -989.9277} C_DIS
LIN {X -1.6722,Y 5.4873,Z 58,A -2.4685,B 0,C 0,E1 0.1598,E2 -989.9277} C_DIS
LIN {X -2.6421,Y 5.0856,Z 58,A -2.5212,B 0,C 0,E1 0.1598,E2 -989.9279} C_DIS
LIN {X -3.3572,Y 4.645,Z 58,A -2.5663,B 0,C 0,E1 0.1598,E2 -989.9279} C_DIS
LIN {X -4.2153,Y 3.8902,Z 58,A -2.6298,B 0,C 0,E1 0.1598,E2 -989.9282} C_DIS
LIN {X -4.7551,Y 3.199,Z 58,A -2.679,B 0,C 0,E1 0.1598,E2 -989.9282} C_DIS
LIN {X -5.1103,Y 2.5938,Z 58,A -2.7178,B 0,C 0,E1 0.1598,E2 -989.9282} C_DIS
LIN {X -5.39,Y 1.9503,Z 58,A -2.7554,B 0,C 0,E1 0.1598,E2 -989.9283} C_DIS
LIN {X -5.5866,Y 1.2766,Z 58,A -2.7912,B 0,C 0,E1 0.1598,E2 -989.9283} C_DIS
LIN {X -5.7021,Y 0.5846,Z 58,A -2.8248,B 0,C 0,E1 0.1598,E2 -989.9284} C_DIS
LIN {X -5.7287,Y -0.1166,Z 58,A -2.8555,B 0,C 0,E1 0.1598,E2 -989.9284} C_DIS
LIN {X -5.6503,Y -0.9902,Z 58,A -2.8895,B 0,C 0,E1 0.1598,E2 -989.9288} C_DIS
LIN {X -5.3318,Y -2.1037,Z 58,A -2.9249,B 0,C 0,E1 0.1598,E2 -989.929} C_DIS
LIN {X -4.996,Y -2.8069,Z 58,A -2.9428,B 0,C 0,E1 0.1598,E2 -989.9286} C_DIS
LIN {X -4.5701,Y -3.4596,Z 58,A -2.955,B 0,C 0,E1 0.1598,E2 -989.9286} C_DIS
LIN {X -4.057,Y -4.0459,Z 58,A -2.9611,B 0,C 0,E1 0.1598,E2 -989.9286} C_DIS
LIN {X -3.4703,Y -4.5586,Z 58,A -2.9614,B 0,C 0,E1 0.1598,E2 -989.9286} C_DIS
LIN {X -2.6518,Y -5.0867,Z 58,A -2.9539,B 0,C 0,E1 0.1598,E2 -989.9286} C_DIS
LIN {X -1.5926,Y -5.5067,Z 58,A -2.933,B 0,C 0,E1 0.1598,E2 -989.9284} C_DIS
LIN {X -0.8704,Y -5.6626,Z 58,A -2.9132,B 0,C 0,E1 0.1598,E2 -989.9284} C_DIS
LIN {X -0.1348,Y -5.7295,Z 58,A -2.8891,B 0,C 0,E1 0.1598,E2 -989.9283} C_DIS
LIN {X -0.1348,Y -5.7295,Z 58,A -2.8891,B 0,C 0,E1 0.1598,E2 -989.9283} C_DIS
Enddeposition()
LIN {X 0.0164,Y -4.7569,Z 58,A -2.8406,B 0,C 0,E1 0.1598,E2 -989.9295} C_DIS
Startdeposition()
$VEL.CP = VEL_PRINT
LIN {X -0.7242,Y -4.7002,Z 58,A -2.8666,B 0,C 0,E1 0.1598,E2 -989.9283} C_DIS
LIN {X -1.4132,Y -4.5399,Z 58,A -2.8851,B 0,C 0,E1 0.1598,E2 -989.9283} C_DIS
LIN {X -2.0718,Y -4.2818,Z 58,A -2.8983,B 0,C 0,E1 0.1598,E2 -989.9283} C_DIS
LIN {X -2.7991,Y -3.8445,Z 58,A -2.9063,B 0,C 0,E1 0.1598,E2 -989.9284} C_DIS
LIN {X -3.3378,Y -3.3861,Z 58,A -2.9065,B 0,C 0,E1 0.1598,E2 -989.9284} C_DIS
LIN {X -3.8032,Y -2.8534,Z 58,A -2.9009,B 0,C 0,E1 0.1598,E2 -989.9284} C_DIS
LIN {X -4.1849,Y -2.2579,Z 58,A -2.8896,B 0,C 0,E1 0.1598,E2 -989.9284} C_DIS
LIN {X -4.498,Y -1.5457,Z 58,A -2.8708,B 0,C 0,E1 0.1598,E2 -989.9285} C_DIS
LIN {X -4.6903,Y -0.7917,Z 58,A -2.8457,B 0,C 0,E1 0.1598,E2 -989.9285} C_DIS
LIN {X -4.7556,Y 0.0544,Z 58,A -2.8121,B 0,C 0,E1 0.1598,E2 -989.9285} C_DIS
LIN {X -4.693,Y 0.759,Z 58,A -2.78,B 0,C 0,E1 0.1598,E2 -989.9285} C_DIS
LIN {X -4.5303,Y 1.4474,Z 58,A -2.7448,B 0,C 0,E1 0.1598,E2 -989.9283} C_DIS
LIN {X -4.2646,Y 2.103,Z 58,A -2.7072,B 0,C 0,E1 0.1598,E2 -989.9283} C_DIS
LIN {X -3.8657,Y 2.7709,Z 58,A -2.6641,B 0,C 0,E1 0.1598,E2 -989.9283} C_DIS
LIN {X -3.4112,Y 3.313,Z 58,A -2.6244,B 0,C 0,E1 0.1598,E2 -989.9281} C_DIS
LIN {X -2.8828,Y 3.7836,Z 58,A -2.585,B 0,C 0,E1 0.1598,E2 -989.928} C_DIS
LIN {X -2.1646,Y 4.2357,Z 58,A -2.5394,B 0,C 0,E1 0.1598,E2 -989.928} C_DIS
LIN {X -1.4449,Y 4.5315,Z 58,A -2.5003,B 0,C 0,E1 0.1598,E2 -989.9278} C_DIS
LIN {X -0.7564,Y 4.6941,Z 58,A -2.4681,B 0,C 0,E1 0.1598,E2 -989.9278} C_DIS
LIN {X 0.0191,Y 4.756,Z 58,A -2.4369,B 0,C 0,E1 0.1598,E2 -989.9277} C_DIS
LIN {X 0.7243,Y 4.7,Z 58,A -2.4133,B 0,C 0,E1 0.1598,E2 -989.9277} C_DIS
LIN {X 1.4138,Y 4.5414,Z 58,A -2.3946,B 0,C 0,E1 0.1598,E2 -989.9277} C_DIS
LIN {X 2.0711,Y 4.2799,Z 58,A -2.3815,B 0,C 0,E1 0.1598,E2 -989.9277} C_DIS
LIN {X 2.742,Y 3.8862,Z 58,A -2.3735,B 0,C 0,E1 0.1598,E2 -989.9277} C_DIS
LIN {X 3.3893,Y 3.3371,Z 58,A -2.3729,B 0,C 0,E1 0.1598,E2 -989.9278} C_DIS
LIN {X 3.8468,Y 2.7973,Z 58,A -2.3791,B 0,C 0,E1 0.1598,E2 -989.9278} C_DIS
LIN {X 4.3133,Y 2.0053,Z 58,A -2.3955,B 0,C 0,E1 0.1598,E2 -989.928} C_DIS
LIN {X 4.5995,Y 1.2065,Z 58,A -2.4191,B 0,C 0,E1 0.1598,E2 -989.928} C_DIS
LIN {X 4.7273,Y 0.5108,Z 58,A -2.4442,B 0,C 0,E1 0.1598,E2 -989.928} C_DIS
LIN {X 4.7476,Y -0.2669,Z 58,A -2.4765,B 0,C 0,E1 0.1598,E2 -989.928} C_DIS
LIN {X 4.6408,Y -1.0375,Z 58,A -2.5134,B 0,C 0,E1 0.1598,E2 -989.928} C_DIS
LIN {X 4.383,Y -1.8459,Z 58,A -2.5574,B 0,C 0,E1 0.1598,E2 -989.9282} C_DIS
LIN {X 4.0229,Y -2.5354,Z 58,A -2.6001,B 0,C 0,E1 0.1598,E2 -989.9282} C_DIS
LIN {X 3.5568,Y -3.1585,Z 58,A -2.6439,B 0,C 0,E1 0.1598,E2 -989.9282} C_DIS
LIN {X 2.9391,Y -3.7404,Z 58,A -2.6915,B 0,C 0,E1 0.1598,E2 -989.9282} C_DIS
LIN {X 2.2271,Y -4.2022,Z 58,A -2.7374,B 0,C 0,E1 0.1598,E2 -989.9282} C_DIS
LIN {X 1.512,Y -4.5085,Z 58,A -2.7768,B 0,C 0,E1 0.1598,E2 -989.9282} C_DIS
LIN {X 0.8263,Y -4.6822,Z 58,A -2.8094,B 0,C 0,E1 0.1598,E2 -989.9282} C_DIS
LIN {X 0.0164,Y -4.7569,Z 58,A -2.8423,B 0,C 0,E1 0.1598,E2 -989.9282} C_DIS
Enddeposition()
LIN {X 0.0164,Y -4.7569,Z 63,A -2.8323,B 0,C 0,E1 0.1598,E2 -989.928} C_DIS
LIN {X 0.0164,Y -4.7567,Z 78,A -2.8068,B 0,C 0,E1 0.1598,E2 -989.9269} C_DIS
LIN {X 0.0164,Y -4.7567,Z 97.1262,A -2.7823,B 0,C 0,E1 0.1598,E2 -989.9267} C_DIS
LIN {X 0.0799,Y -43.69,Z 97.1262,A -96.8823,B 24.8469,C -2.855,E1 25,E2 -900.2489} C_DIS
LIN {X 0.0799,Y -43.69,Z 77.1262,A -96.5524,B 24.8614,C -2.7164,E1 25,E2 -900.2489} C_DIS
LIN {X 0.0924,Y -37.3508,Z 63.5315,A -96.5891,B 24.8598,C -2.7318,E1 25,E2 -900.2489} C_DIS
LIN {X 0.0966,Y -35.2377,Z 59,A -96.6028,B 24.8592,C -2.7375,E1 25,E2 -900.2489} C_DIS
Startdeposition()
$VEL.CP = VEL_PRINT
LIN {X -1.7292,Y -35.1988,Z 59,A -100.1544,B 24.86,C -2.7302,E1 24.99,E2 -896.6792} C_DIS
LIN {X -3.8843,Y -35.026,Z 59,A -103.6526,B 24.86,C -2.7306,E1 24.9803,E2 -893.1802} C_DIS
LIN {X -6.0249,Y -34.7223,Z 59,A -107.3189,B 24.86,C -2.7298,E1 24.9702,E2 -889.5086} C_DIS
LIN {X -8.384,Y -34.2289,Z 59,A -111.1873,B 24.8598,C -2.7322,E1 24.9596,E2 -885.641} C_DIS
LIN {X -10.643,Y -33.5954,Z 59,A -114.9746,B 24.8595,C -2.7351,E1 24.9495,E2 -881.8543} C_DIS
LIN {X -12.7423,Y -32.8567,Z 59,A -118.6094,B 24.8592,C -2.7381,E1 24.94,E2 -878.2191} C_DIS
LIN {X -14.8426,Y -31.9626,Z 59,A -122.307,B 24.8588,C -2.7422,E1 24.9306,E2 -874.5224} C_DIS
LIN {X -16.8882,Y -30.9306,Z 59,A -126.0576,B 24.8583,C -2.7466,E1 24.9213,E2 -870.772} C_DIS
LIN {X -18.8224,Y -29.7935,Z 59,A -129.7618,B 24.8578,C -2.7512,E1 24.9125,E2 -867.0673} C_DIS
LIN {X -20.715,Y -28.5099,Z 59,A -133.4984,B 24.8572,C -2.757,E1 24.9039,E2 -863.3318} C_DIS
LIN {X -22.4875,Y -27.1334,Z 59,A -137.1188,B 24.8565,C -2.7638,E1 24.896,E2 -859.7141} C_DIS
LIN {X -24.2659,Y -25.5559,Z 59,A -140.9496,B 24.8557,C -2.7717,E1 24.8882,E2 -855.8866} C_DIS
LIN {X -25.8004,Y -24.0059,Z 59,A -144.4937,B 24.8549,C -2.7791,E1 24.8813,E2 -852.345} C_DIS
LIN {X -27.2156,Y -22.3886,Z 59,A -148.1077,B 24.8542,C -2.7858,E1 24.8748,E2 -848.7305} C_DIS
LIN {X -28.6009,Y -20.5893,Z 59,A -151.8008,B 24.8533,C -2.7946,E1 24.8686,E2 -845.0406} C_DIS
LIN {X -29.861,Y -18.7145,Z 59,A -155.4649,B 24.8523,C -2.8039,E1 24.8631,E2 -841.3802} C_DIS
LIN {X -31.0371,Y -16.6919,Z 59,A -159.3343,B 24.8513,C -2.8133,E1 24.8578,E2 -837.5129} C_DIS
LIN {X -32.0398,Y -14.6753,Z 59,A -163.0292,B 24.8503,C -2.8229,E1 24.8533,E2 -833.8212} C_DIS
LIN {X -32.9248,Y -12.5648,Z 59,A -166.7771,B 24.8492,C -2.8332,E1 24.8494,E2 -830.0769} C_DIS
LIN {X -33.6898,Y -10.34,Z 59,A -170.5742,B 24.848,C -2.8445,E1 24.8462,E2 -826.2852} C_DIS
LIN {X -34.2872,Y -8.1427,Z 59,A -174.3188,B 24.8468,C -2.8552,E1 24.8436,E2 -822.5442} C_DIS
LIN {X -34.7261,Y -6.0038,Z 59,A -177.9925,B 24.8458,C -2.8649,E1 24.8417,E2 -818.872} C_DIS
LIN {X -35.0413,Y -3.7442,Z 59,A 178.3432,B 24.8445,C -2.8767,E1 24.8404,E2 -815.214} C_DIS
LIN {X -35.2131,Y -1.3992,Z 59,A 174.5032,B 24.8432,C -2.8884,E1 24.8398,E2 -811.3789} C_DIS
LIN {X -35.2323,Y 0.7822,Z 59,A 170.9224,B 24.8421,C -2.8992,E1 24.8398,E2 -807.8024} C_DIS
LIN {X -35.1139,Y 2.9922,Z 59,A 167.2758,B 24.8409,C -2.91,E1 24.8406,E2 -804.1598} C_DIS
LIN {X -34.8572,Y 5.1885,Z 59,A 163.5951,B 24.8397,C -2.9205,E1 24.842,E2 -800.4824} C_DIS
LIN {X -34.4413,Y 7.4637,Z 59,A 159.905,B 24.8384,C -2.9328,E1 24.844,E2 -796.7998} C_DIS
LIN {X -33.8805,Y 9.6968,Z 59,A 156.0906,B 24.8372,C -2.9437,E1 24.8467,E2 -792.9893} C_DIS
LIN {X -33.1806,Y 11.8722,Z 59,A 152.4058,B 24.8359,C -2.9552,E1 24.85,E2 -789.3109} C_DIS
LIN {X -32.3583,Y 13.9594,Z 59,A 148.7122,B 24.8347,C -2.9656,E1 24.854,E2 -785.6217} C_DIS
LIN {X -31.4185,Y 15.9622,Z 59,A 145.1028,B 24.8336,C -2.9759,E1 24.8584,E2 -782.0175} C_DIS
LIN {X -30.3288,Y 17.9464,Z 59,A 141.4084,B 24.8324,C -2.9861,E1 24.8635,E2 -778.3282} C_DIS
LIN {X -29.0651,Y 19.9292,Z 59,A 137.5861,B 24.8312,C -2.9965,E1 24.8693,E2 -774.5116} C_DIS
LIN {X -27.7845,Y 21.6789,Z 59,A 133.9571,B 24.8303,C -3.0048,E1 24.8754,E2 -770.885} C_DIS
LIN {X -26.3271,Y 23.4266,Z 59,A 130.2748,B 24.8292,C -3.0142,E1 24.8821,E2 -767.2085} C_DIS
LIN {X -24.8277,Y 25.01,Z 59,A 126.7162,B 24.8283,C -3.0224,E1 24.8891,E2 -763.6544} C_DIS
LIN {X -23.2558,Y 26.478,Z 59,A 123.1972,B 24.8274,C -3.0301,E1 24.8964,E2 -760.1396} C_DIS
LIN {X -21.499,Y 27.9232,Z 59,A 119.484,B 24.8265,C -3.0377,E1 24.9044,E2 -756.4308} C_DIS
LIN {X -19.6606,Y 29.2469,Z 59,A 115.7655,B 24.8258,C -3.0445,E1 24.913,E2 -752.7159} C_DIS
LIN {X -17.7453,Y 30.4475,Z 59,A 112.0038,B 24.8251,C -3.0502,E1 24.9219,E2 -748.9562} C_DIS
LIN {X -15.6798,Y 31.5603,Z 59,A 108.2676,B 24.8243,C -3.0571,E1 24.9312,E2 -745.2263} C_DIS
LIN {X -13.6073,Y 32.5078,Z 59,A 104.5396,B 24.8237,C -3.0622,E1 24.9407,E2 -741.5016} C_DIS
LIN {X -11.4642,Y 33.324,Z 59,A 100.7501,B 24.8233,C -3.0662,E1 24.9507,E2 -737.7141} C_DIS
LIN {X -9.2857,Y 33.9955,Z 59,A 97.0363,B 24.8228,C -3.07,E1 24.9606,E2 -734.0033} C_DIS
LIN {X -7.0557,Y 34.5272,Z 59,A 93.4164,B 24.8223,C -3.0744,E1 24.9705,E2 -730.3893} C_DIS
LIN {X -4.7821,Y 34.9152,Z 59,A 89.6332,B 24.8221,C -3.0766,E1 24.9809,E2 -726.6078} C_DIS
LIN {X -2.5925,Y 35.1454,Z 59,A 86.0795,B 24.8218,C -3.0785,E1 24.9908,E2 -723.0571} C_DIS
LIN {X -0.3902,Y 35.239,Z 59,A 82.373,B 24.8218,C -3.0782,E1 25.0011,E2 -719.3492} C_DIS
LIN {X 1.9132,Y 35.1888,Z 59,A 78.7303,B 24.8218,C -3.0796,E1 25.0113,E2 -715.711} C_DIS
LIN {X 4.1309,Y 34.9978,Z 59,A 75.1276,B 24.8218,C -3.0794,E1 25.0213,E2 -712.11} C_DIS
LIN {X 6.4126,Y 34.6528,Z 59,A 71.3238,B 24.8219,C -3.0776,E1 25.0317,E2 -708.3057} C_DIS
LIN {X 8.5628,Y 34.1847,Z 59,A 67.6916,B 24.8222,C -3.075,E1 25.0416,E2 -704.6727} C_DIS
LIN {X 10.8184,Y 33.5391,Z 59,A 63.9529,B 24.8224,C -3.0732,E1 25.0516,E2 -700.9363} C_DIS
LIN {X 12.9142,Y 32.7892,Z 59,A 60.3165,B 24.8229,C -3.0697,E1 25.0611,E2 -697.2992} C_DIS
LIN {X 14.9913,Y 31.8933,Z 59,A 56.6672,B 24.8233,C -3.066,E1 25.0704,E2 -693.6502} C_DIS
LIN {X 16.9737,Y 30.8843,Z 59,A 53.011,B 24.8239,C -3.0608,E1 25.0794,E2 -689.992} C_DIS
LIN {X 18.9052,Y 29.741,Z 59,A 49.3276,B 24.8245,C -3.055,E1 25.0882,E2 -686.3065} C_DIS
LIN {X 20.7727,Y 28.4676,Z 59,A 45.7558,B 24.8251,C -3.0504,E1 25.0964,E2 -682.736} C_DIS
LIN {X 22.5636,Y 27.0702,Z 59,A 42.0509,B 24.8259,C -3.0436,E1 25.1044,E2 -679.0289} C_DIS
LIN {X 24.2659,Y 25.5559,Z 59,A 38.4182,B 24.8266,C -3.0373,E1 25.1119,E2 -675.3959} C_DIS
LIN {X 25.8004,Y 24.0059,Z 59,A 34.9085,B 24.8274,C -3.0303,E1 25.1187,E2 -671.8848} C_DIS
LIN {X 27.2156,Y 22.3886,Z 59,A 31.332,B 24.8284,C -3.0212,E1 25.1252,E2 -668.3032} C_DIS
LIN {X 28.6009,Y 20.5893,Z 59,A 27.6794,B 24.8294,C -3.013,E1 25.1312,E2 -664.6485} C_DIS
LIN {X 29.861,Y 18.7145,Z 59,A 24.0575,B 24.8303,C -3.0045,E1 25.1368,E2 -661.0246} C_DIS
LIN {X 31.0371,Y 16.6919,Z 59,A 20.2348,B 24.8315,C -2.9942,E1 25.142,E2 -657.1976} C_DIS
LIN {X 32.0398,Y 14.6753,Z 59,A 16.5863,B 24.8326,C -2.9844,E1 25.1464,E2 -653.5455} C_DIS
LIN {X 32.9248,Y 12.5648,Z 59,A 12.8872,B 24.8337,C -2.9742,E1 25.1502,E2 -649.8426} C_DIS
LIN {X 33.6898,Y 10.34,Z 59,A 9.141,B 24.8349,C -2.9643,E1 25.1535,E2 -646.094} C_DIS
LIN {X 34.2872,Y 8.1427,Z 59,A 5.4475,B 24.8361,C -2.9534,E1 25.156,E2 -642.396} C_DIS
LIN {X 34.7261,Y 6.0038,Z 59,A 1.8251,B 24.8374,C -2.9415,E1 25.1579,E2 -638.7668} C_DIS
LIN {X 35.0413,Y 3.7442,Z 59,A -1.7874,B 24.8385,C -2.9315,E1 25.1591,E2 -635.152} C_DIS
LIN {X 35.2115,Y 1.4363,Z 59,A -5.5412,B 24.8398,C -2.92,E1 25.1597,E2 -631.3931} C_DIS
LIN {X 35.2363,Y -0.5608,Z 59,A -8.7404,B 24.8408,C -2.9105,E1 25.1597,E2 -628.1906} C_DIS
LIN {X 35.132,Y -2.7656,Z 59,A -12.2912,B 24.842,C -2.8998,E1 25.1591,E2 -624.6356} C_DIS
LIN {X 34.8949,Y -4.9252,Z 59,A -15.7682,B 24.8431,C -2.8896,E1 25.1579,E2 -621.1549} C_DIS
LIN {X 34.491,Y -7.2318,Z 59,A -19.6371,B 24.8445,C -2.8768,E1 25.1558,E2 -617.2783} C_DIS
LIN {X 33.9311,Y -9.5182,Z 59,A -23.4152,B 24.8457,C -2.8658,E1 25.1531,E2 -613.4958} C_DIS
LIN {X 33.2423,Y -11.6986,Z 59,A -27.0464,B 24.8468,C -2.8558,E1 25.1499,E2 -609.8615} C_DIS
LIN {X 32.4336,Y -13.7833,Z 59,A -30.7169,B 24.848,C -2.8444,E1 25.1461,E2 -606.1843} C_DIS
LIN {X 31.478,Y -15.8447,Z 59,A -34.3955,B 24.8491,C -2.8339,E1 25.1416,E2 -602.5006} C_DIS
LIN {X 30.3785,Y -17.8623,Z 59,A -38.0801,B 24.8502,C -2.824,E1 25.1365,E2 -598.8118} C_DIS
LIN {X 29.1202,Y -19.8477,Z 59,A -41.8266,B 24.8512,C -2.8147,E1 25.1308,E2 -595.0618} C_DIS
LIN {X 27.7845,Y -21.6789,Z 59,A -45.5656,B 24.8523,C -2.8042,E1 25.1245,E2 -591.3158} C_DIS
LIN {X 26.3271,Y -23.4266,Z 59,A -49.2053,B 24.8532,C -2.7957,E1 25.1178,E2 -587.6726} C_DIS
LIN {X 24.8277,Y -25.01,Z 59,A -52.7248,B 24.854,C -2.7876,E1 25.111,E2 -584.149} C_DIS
LIN {X 23.2558,Y -26.478,Z 59,A -56.2073,B 24.8548,C -2.7799,E1 25.1038,E2 -580.6622} C_DIS
LIN {X 21.499,Y -27.9232,Z 59,A -59.8844,B 24.8556,C -2.7723,E1 25.0957,E2 -576.9809} C_DIS
LIN {X 19.6606,Y -29.2469,Z 59,A -63.5693,B 24.8564,C -2.765,E1 25.0873,E2 -573.2914} C_DIS
LIN {X 17.7453,Y -30.4475,Z 59,A -67.2998,B 24.8572,C -2.7576,E1 25.0783,E2 -569.5549} C_DIS
LIN {X 15.6798,Y -31.5603,Z 59,A -71.0081,B 24.8577,C -2.7528,E1 25.0691,E2 -565.8455} C_DIS
LIN {X 13.6073,Y -32.5078,Z 59,A -74.7111,B 24.8582,C -2.7474,E1 25.0597,E2 -562.1386} C_DIS
LIN {X 11.4642,Y -33.324,Z 59,A -78.4784,B 24.8588,C -2.7421,E1 25.0498,E2 -558.3666} C_DIS
LIN {X 9.2857,Y -33.9955,Z 59,A -82.1739,B 24.8592,C -2.7382,E1 25.0398,E2 -554.6681} C_DIS
LIN {X 7.0557,Y -34.5272,Z 59,A -85.779,B 24.8594,C -2.7364,E1 25.03,E2 -551.0635} C_DIS
LIN {X 4.7821,Y -34.9152,Z 59,A -89.5502,B 24.8597,C -2.7335,E1 25.0196,E2 -547.289} C_DIS
LIN {X 2.5925,Y -35.1454,Z 59,A -93.0958,B 24.8598,C -2.7321,E1 25.0097,E2 -543.7421} C_DIS
LIN {X 0.4325,Y -35.2383,Z 59,A -96.5877,B 24.8598,C -2.7312,E1 25,E2 -540.2489} C_DIS
LIN {X 0.4325,Y -35.2383,Z 59,A -96.5877,B 24.8598,C -2.7312,E1 25,E2 -540.2489} C_DIS
Enddeposition()
LIN {X 0.0839,Y -34.2576,Z 59,A -95.8072,B 24.8565,C -2.7643,E1 25.0024,E2 -541.108} C_DIS
Startdeposition()
$VEL.CP = VEL_PRINT
LIN {X 2.02,Y -34.2004,Z 59,A -92.6026,B 24.8565,C -2.765,E1 25.0113,E2 -544.3134} C_DIS
LIN {X 3.8572,Y -34.0423,Z 59,A -89.1276,B 24.8557,C -2.7714,E1 25.021,E2 -547.8014} C_DIS
LIN {X 6.2267,Y -33.6898,Z 59,A -85.2675,B 24.8557,C -2.7725,E1 25.0317,E2 -551.6603} C_DIS
LIN {X 8.2797,Y -33.2445,Z 59,A -81.6839,B 24.8552,C -2.7767,E1 25.0414,E2 -555.2488} C_DIS
LIN {X 10.4184,Y -32.6377,Z 59,A -77.9126,B 24.8547,C -2.7816,E1 25.0515,E2 -559.025} C_DIS
LIN {X 12.2302,Y -32.0027,Z 59,A -74.9759,B 24.8547,C -2.7821,E1 25.0592,E2 -561.9569} C_DIS
Enddeposition()
END
